  MoveL 10820 to (-38.97, 156.79, 153.89) mm, rotated rx -180 ry 0 rz 180 deg; joints [-53.214, -19.541, 102.145, 84.502, 53.57, -80.793]
  Call Extruder(791.10708)
  Set speed (40.0 mm/s)
  MoveL 10821 to (-38.97, 156.79, 153.89) mm, rotated rx -180 ry 0 rz 180 deg; joints [-53.214, -19.541, 102.145, 84.502, 53.57, -80.793]
  Call Extruder(0.00000)
  Set speed (130.0 mm/s)
  MoveL 10822 to (-31.64, 163.21, 153.89) mm, rotated rx 180 ry 0 rz 180 deg; joints [-52.884, -18.131, 101.16, 84.753, 53.204, -81.283]
  Call Extruder(2.00000)
  Set speed (40.0 mm/s)
  MoveL 10823 to (-31.64, 163.21, 153.89) mm, rotated rx 180 ry 0 rz 180 deg; joints [-52.884, -18.131, 101.16, 84.753, 53.204, -81.283]
  Set speed (30.0 mm/s)
  MoveL 10824 to (-31.64, 163.21, 153.89) mm, rotated rx 180 ry 0 rz 180 deg; joints [-52.884, -18.131, 101.16, 84.753, 53.204, -81.283]
  Call Extruder(2.18198)
  MoveL 10825 to (-31.93, 163.09, 153.89) mm, rotated rx 180 ry 0 rz 180 deg; joints [-52.91, -18.171, 101.189, 84.749, 53.231, -81.271]
  MoveL 10826 to (-31.93, 163.09, 153.89) mm, rotated rx 180 ry 0 rz 180 deg; joints [-52.91, -18.171, 101.189, 84.749, 53.231, -81.271]
  Call Extruder(2.36471)
  MoveL 10827 to (-32.22, 162.97, 153.89) mm, rotated rx -180 ry 0 rz -180 deg; joints [-52.936, -18.212, 101.218, 84.745, 53.257, -81.26]
  MoveL 10828 to (-32.22, 162.97, 153.89) mm, rotated rx -180 ry 0 rz -180 deg; joints [-52.936, -18.212, 101.218, 84.745, 53.257, -81.26]
  Call Extruder(2.53265)
  MoveL 10829 to (-32.49, 162.85, 153.89) mm, rotated rx 180 ry 0 rz 180 deg; joints [-52.96, -18.249, 101.244, 84.742, 53.282, -81.249]
  MoveL 10830 to (-32.49, 162.85, 153.89) mm, rotated rx 180 ry 0 rz 180 deg; joints [-52.96, -18.249, 101.244, 84.742, 53.282, -81.249]
  Call Extruder(2.68564)
  MoveL 10831 to (-32.73, 162.75, 153.89) mm, rotated rx -180 ry 0 rz 180 deg; joints [-52.981, -18.282, 101.268, 84.738, 53.304, -81.239]
  MoveL 10832 to (-32.73, 162.75, 153.89) mm, rotated rx -180 ry 0 rz 180 deg; joints [-52.981, -18.282, 101.268, 84.738, 53.304, -81.239]
  Call Extruder(2.83919)
  MoveL 10833 to (-32.97, 162.65, 153.89) mm, rotated rx 180 ry 0 rz 180 deg; joints [-53.002, -18.316, 101.292, 84.735, 53.326, -81.229]
  MoveL 10834 to (-32.97, 162.65, 153.89) mm, rotated rx 180 ry 0 rz 180 deg; joints [-53.002, -18.316, 101.292, 84.735, 53.326, -81.229]
  Call Extruder(3.04828)
  MoveL 10835 to (-33.28, 162.47, 153.89) mm, rotated rx -180 ry 0 rz 180 deg; joints [-53.025, -18.365, 101.326, 84.729, 53.349, -81.214]
  MoveL 10836 to (-33.28, 162.47, 153.89) mm, rotated rx -180 ry 0 rz 180 deg; joints [-53.025, -18.365, 101.326, 84.729, 53.349, -81.214]
  Call Extruder(3.25817)
  MoveL 10837 to (-33.59, 162.29, 153.89) mm, rotated rx 180 ry 0 rz 180 deg; joints [-53.048, -18.413, 101.36, 84.723, 53.373, -81.199]
  MoveL 10838 to (-33.59, 162.29, 153.89) mm, rotated rx 180 ry 0 rz 180 deg; joints [-53.048, -18.413, 101.36, 84.723, 53.373, -81.199]
  Call Extruder(3.46884)
  MoveL 10839 to (-33.9, 162.11, 153.89) mm, rotated rx 180 ry 0 rz 180 deg; joints [-53.07, -18.462, 101.394, 84.716, 53.397, -81.184]
  MoveL 10840 to (-33.9, 162.11, 153.89) mm, rotated rx 180 ry 0 rz 180 deg; joints [-53.07, -18.462, 101.394, 84.716, 53.397, -81.184]
  Call Extruder(3.68030)
  MoveL 10841 to (-34.2, 161.93, 153.89) mm, rotated rx -180 ry 0 rz 180 deg; joints [-53.093, -18.51, 101.428, 84.71, 53.421, -81.169]
  MoveL 10842 to (-34.2, 161.93, 153.89) mm, rotated rx -180 ry 0 rz 180 deg; joints [-53.093, -18.51, 101.428, 84.71, 53.421, -81.169]
  Call Extruder(3.88506)
  MoveL 10843 to (-34.49, 161.74, 153.89) mm, rotated rx 180 ry 0 rz -180 deg; joints [-53.111, -18.558, 101.462, 84.703, 53.439, -81.153]
  MoveL 10844 to (-34.49, 161.74, 153.89) mm, rotated rx 180 ry 0 rz -180 deg; joints [-53.111, -18.558, 101.462, 84.703, 53.439, -81.153]
  Call Extruder(4.20602)
  MoveL 10845 to (-34.92, 161.42, 153.89) mm, rotated rx 180 ry 0 rz 180 deg; joints [-53.137, -18.634, 101.516, 84.691, 53.467, -81.128]
  MoveL 10846 to (-34.92, 161.42, 153.89) mm, rotated rx 180 ry 0 rz 180 deg; joints [-53.137, -18.634, 101.516, 84.691, 53.467, -81.128]
  Call Extruder(4.52807)
  MoveL 10847 to (-35.35, 161.1, 153.89) mm, rotated rx 180 ry 0 rz -180 deg; joints [-53.163, -18.71, 101.569, 84.679, 53.495, -81.103]
  Call Extruder(5.35599)
  MoveL 10848 to (-36.39, 160.19, 153.89) mm, rotated rx 180 ry 0 rz 180 deg; joints [-53.209, -18.91, 101.708, 84.644, 53.547, -81.033]
  Call Extruder(6.18392)
  MoveL 10849 to (-37.3, 159.15, 153.89) mm, rotated rx -180 ry 0 rz 180 deg; joints [-53.227, -19.113, 101.85, 84.602, 53.57, -80.959]
  Call Extruder(6.34862)
  MoveL 10850 to (-37.46, 158.93, 153.89) mm, rotated rx -180 ry 0 rz 180 deg; joints [-53.227, -19.154, 101.878, 84.593, 53.571, -80.943]
  MoveL 10851 to (-37.46, 158.93, 153.89) mm, rotated rx -180 ry 0 rz 180 deg; joints [-53.227, -19.154, 101.878, 84.593, 53.571, -80.943]
  Call Extruder(6.67688)
  MoveL 10852 to (-37.79, 158.49, 153.89) mm, rotated rx -180 ry 0 rz 180 deg; joints [-53.226, -19.235, 101.934, 84.574, 53.572, -80.912]
  MoveL 10853 to (-37.79, 158.49, 153.89) mm, rotated rx -180 ry 0 rz 180 deg; joints [-53.226, -19.235, 101.934, 84.574, 53.572, -80.912]
  Call Extruder(7.00398)
  MoveL 10854 to (-38.11, 158.04, 153.89) mm, rotated rx 180 ry 0 rz 180 deg; joints [-53.224, -19.316, 101.99, 84.556, 53.573, -80.881]
  MoveL 10855 to (-38.11, 158.04, 153.89) mm, rotated rx 180 ry 0 rz 180 deg; joints [-53.224, -19.316, 101.99, 84.556, 53.573, -80.881]
  Call Extruder(7.13851)
  MoveL 10856 to (-38.23, 157.85, 153.89) mm, rotated rx -180 ry 0 rz 180 deg; joints [-53.22, -19.35, 102.013, 84.547, 53.57, -80.868]
  MoveL 10857 to (-38.23, 157.85, 153.89) mm, rotated rx -180 ry 0 rz 180 deg; joints [-53.22, -19.35, 102.013, 84.547, 53.57, -80.868]
  Call Extruder(7.35382)
  MoveL 10858 to (-38.41, 157.53, 153.89) mm, rotated rx 180 ry 0 rz 180 deg; joints [-53.213, -19.403, 102.05, 84.534, 53.564, -80.847]
  MoveL 10859 to (-38.41, 157.53, 153.89) mm, rotated rx 180 ry 0 rz 180 deg; joints [-53.213, -19.403, 102.05, 84.534, 53.564, -80.847]
  Call Extruder(7.56829)
  MoveL 10860 to (-38.59, 157.22, 153.89) mm, rotated rx 180 ry 0 rz 180 deg; joints [-53.205, -19.456, 102.087, 84.52, 53.559, -80.825]
  MoveL 10861 to (-38.59, 157.22, 153.89) mm, rotated rx 180 ry 0 rz 180 deg; joints [-53.205, -19.456, 102.087, 84.52, 53.559, -80.825]
  Call Extruder(7.78192)
  MoveL 10862 to (-38.77, 156.9, 153.89) mm, rotated rx 180 ry 0 rz 180 deg; joints [-53.198, -19.51, 102.123, 84.506, 53.553, -80.804]
  MoveL 10863 to (-38.77, 156.9, 153.89) mm, rotated rx 180 ry 0 rz 180 deg; joints [-53.198, -19.51, 102.123, 84.506, 53.553, -80.804]
  Call Extruder(7.96114)
  MoveL 10864 to (-38.91, 156.63, 153.89) mm, rotated rx 180 ry 0 rz 180 deg; joints [-53.189, -19.554, 102.154, 84.494, 53.546, -80.786]
  MoveL 10865 to (-38.91, 156.63, 153.89) mm, rotated rx 180 ry 0 rz 180 deg; joints [-53.189, -19.554, 102.154, 84.494, 53.546, -80.786]
  Call Extruder(8.10685)
  MoveL 10866 to (-39.01, 156.4, 153.89) mm, rotated rx -180 ry 0 rz 180 deg; joints [-53.18, -19.59, 102.179, 84.484, 53.537, -80.771]
  MoveL 10867 to (-39.01, 156.4, 153.89) mm, rotated rx -180 ry 0 rz 180 deg; joints [-53.18, -19.59, 102.179, 84.484, 53.537, -80.771]
  Call Extruder(8.25205)
  MoveL 10868 to (-39.1, 156.17, 153.89) mm, rotated rx -180 ry 0 rz 180 deg; joints [-53.17, -19.626, 102.203, 84.474, 53.528, -80.755]
  MoveL 10869 to (-39.1, 156.17, 153.89) mm, rotated rx -180 ry 0 rz 180 deg; joints [-53.17, -19.626, 102.203, 84.474, 53.528, -80.755]
  Call Extruder(8.43477)
  MoveL 10870 to (-39.23, 155.88, 153.89) mm, rotated rx 180 ry 0 rz 180 deg; joints [-53.156, -19.671, 102.234, 84.461, 53.517, -80.736]
  MoveL 10871 to (-39.23, 155.88, 153.89) mm, rotated rx 180 ry 0 rz 180 deg; joints [-53.156, -19.671, 102.234, 84.461, 53.517, -80.736]
  Call Extruder(8.61673)
  MoveL 10872 to (-39.35, 155.58, 153.89) mm, rotated rx 180 ry 0 rz 180 deg; joints [-53.143, -19.716, 102.265, 84.448, 53.505, -80.717]
  MoveL 10873 to (-39.35, 155.58, 153.89) mm, rotated rx 180 ry 0 rz 180 deg; joints [-53.143, -19.716, 102.265, 84.448, 53.505, -80.717]
  Call Extruder(8.76407)
  MoveL 10874 to (-39.44, 155.34, 153.89) mm, rotated rx 180 ry 0 rz -180 deg; joints [-53.131, -19.753, 102.29, 84.437, 53.495, -80.701]
  MoveL 10875 to (-39.44, 155.34, 153.89) mm, rotated rx 180 ry 0 rz -180 deg; joints [-53.131, -19.753, 102.29, 84.437, 53.495, -80.701]
  Call Extruder(8.87730)
  MoveL 10876 to (-39.5, 155.15, 153.89) mm, rotated rx 180 ry 0 rz -180 deg; joints [-53.121, -19.78, 102.309, 84.428, 53.485, -80.689]
  MoveL 10877 to (-39.5, 155.15, 153.89) mm, rotated rx 180 ry 0 rz -180 deg; joints [-53.121, -19.78, 102.309, 84.428, 53.485, -80.689]
  Call Extruder(8.99009)
  MoveL 10878 to (-39.56, 154.97, 153.89) mm, rotated rx 180 ry 0 rz 180 deg; joints [-53.11, -19.808, 102.328, 84.419, 53.475, -80.677]
  MoveL 10879 to (-39.56, 154.97, 153.89) mm, rotated rx 180 ry 0 rz 180 deg; joints [-53.11, -19.808, 102.328, 84.419, 53.475, -80.677]
  Call Extruder(9.10244)
  MoveL 10880 to (-39.62, 154.78, 153.89) mm, rotated rx 180 ry 0 rz 180 deg; joints [-53.099, -19.836, 102.347, 84.411, 53.465, -80.665]
  MoveL 10881 to (-39.62, 154.78, 153.89) mm, rotated rx 180 ry 0 rz 180 deg; joints [-53.099, -19.836, 102.347, 84.411, 53.465, -80.665]
  Call Extruder(9.21434)
  MoveL 10882 to (-39.68, 154.59, 153.89) mm, rotated rx 180 ry 0 rz 180 deg; joints [-53.088, -19.863, 102.366, 84.402, 53.455, -80.653]
  MoveL 10883 to (-39.68, 154.59, 153.89) mm, rotated rx 180 ry 0 rz 180 deg; joints [-53.088, -19.863, 102.366, 84.402, 53.455, -80.653]
  Call Extruder(9.33574)
  MoveL 10884 to (-39.75, 154.38, 153.89) mm, rotated rx -180 ry 0 rz 180 deg; joints [-53.076, -19.893, 102.386, 84.393, 53.444, -80.639]
  MoveL 10885 to (-39.75, 154.38, 153.89) mm, rotated rx -180 ry 0 rz 180 deg; joints [-53.076, -19.893, 102.386, 84.393, 53.444, -80.639]
  Call Extruder(9.46653)
  MoveL 10886 to (-39.81, 154.16, 153.89) mm, rotated rx 180 ry 0 rz 180 deg; joints [-53.063, -19.926, 102.408, 84.382, 53.432, -80.625]
  MoveL 10887 to (-39.81, 154.16, 153.89) mm, rotated rx 180 ry 0 rz 180 deg; joints [-53.063, -19.926, 102.408, 84.382, 53.432, -80.625]
  Call Extruder(9.59676)
  MoveL 10888 to (-39.88, 153.94, 153.89) mm, rotated rx 180 ry 0 rz -180 deg; joints [-53.049, -19.958, 102.43, 84.372, 53.42, -80.611]
  MoveL 10889 to (-39.88, 153.94, 153.89) mm, rotated rx 180 ry 0 rz -180 deg; joints [-53.049, -19.958, 102.43, 84.372, 53.42, -80.611]
  Call Extruder(9.72643)
  MoveL 10890 to (-39.95, 153.71, 153.89) mm, rotated rx 180 ry 0 rz 180 deg; joints [-53.036, -19.99, 102.452, 84.362, 53.407, -80.596]
  MoveL 10891 to (-39.95, 153.71, 153.89) mm, rotated rx 180 ry 0 rz 180 deg; joints [-53.036, -19.99, 102.452, 84.362, 53.407, -80.596]
  Call Extruder(9.85553)
  MoveL 10892 to (-40.02, 153.49, 153.89) mm, rotated rx 180 ry 0 rz 180 deg; joints [-53.022, -20.023, 102.474, 84.351, 53.395, -80.582]
  MoveL 10893 to (-40.02, 153.49, 153.89) mm, rotated rx 180 ry 0 rz 180 deg; joints [-53.022, -20.023, 102.474, 84.351, 53.395, -80.582]
  Call Extruder(9.97061)
  MoveL 10894 to (-40.06, 153.28, 153.89) mm, rotated rx -180 ry 0 rz 180 deg; joints [-53.007, -20.051, 102.493, 84.341, 53.381, -80.569]
  MoveL 10895 to (-40.06, 153.28, 153.89) mm, rotated rx -180 ry 0 rz 180 deg; joints [-53.007, -20.051, 102.493, 84.341, 53.381, -80.569]
  Call Extruder(10.08525)
  MoveL 10896 to (-40.11, 153.08, 153.89) mm, rotated rx -180 ry 0 rz 180 deg; joints [-52.993, -20.079, 102.512, 84.332, 53.368, -80.556]
  MoveL 10897 to (-40.11, 153.08, 153.89) mm, rotated rx -180 ry 0 rz 180 deg; joints [-52.993, -20.079, 102.512, 84.332, 53.368, -80.556]
  Call Extruder(10.19943)
  MoveL 10898 to (-40.15, 152.88, 153.89) mm, rotated rx 180 ry 0 rz 180 deg; joints [-52.978, -20.107, 102.531, 84.322, 53.354, -80.543]
  MoveL 10899 to (-40.15, 152.88, 153.89) mm, rotated rx 180 ry 0 rz 180 deg; joints [-52.978, -20.107, 102.531, 84.322, 53.354, -80.543]
  Call Extruder(10.31316)
  MoveL 10900 to (-40.2, 152.67, 153.89) mm, rotated rx 180 ry 0 rz -180 deg; joints [-52.963, -20.135, 102.55, 84.312, 53.34, -80.53]
  MoveL 10901 to (-40.2, 152.67, 153.89) mm, rotated rx 180 ry 0 rz -180 deg; joints [-52.963, -20.135, 102.55, 84.312, 53.34, -80.53]
  Call Extruder(10.43859)
  MoveL 10902 to (-40.24, 152.45, 153.89) mm, rotated rx -180 ry 0 rz 180 deg; joints [-52.946, -20.166, 102.571, 84.302, 53.325, -80.515]
  MoveL 10903 to (-40.24, 152.45, 153.89) mm, rotated rx -180 ry 0 rz 180 deg; joints [-52.946, -20.166, 102.571, 84.302, 53.325, -80.515]
  Call Extruder(10.57556)
  MoveL 10904 to (-40.29, 152.2, 153.89) mm, rotated rx -180 ry 0 rz 180 deg; joints [-52.928, -20.199, 102.594, 84.29, 53.308, -80.5]
  MoveL 10905 to (-40.29, 152.2, 153.89) mm, rotated rx -180 ry 0 rz 180 deg; joints [-52.928, -20.199, 102.594, 84.29, 53.308, -80.5]
  Call Extruder(10.71193)
  MoveL 10906 to (-40.34, 151.95, 153.89) mm, rotated rx 180 ry 0 rz 180 deg; joints [-52.909, -20.233, 102.617, 84.278, 53.29, -80.484]
  MoveL 10907 to (-40.34, 151.95, 153.89) mm, rotated rx 180 ry 0 rz 180 deg; joints [-52.909, -20.233, 102.617, 84.278, 53.29, -80.484]
  Call Extruder(10.84768)
  MoveL 10908 to (-40.39, 151.7, 153.89) mm, rotated rx -180 ry 0 rz 180 deg; joints [-52.89, -20.267, 102.639, 84.266, 53.273, -80.468]
  MoveL 10909 to (-40.39, 151.7, 153.89) mm, rotated rx -180 ry 0 rz 180 deg; joints [-52.89, -20.267, 102.639, 84.266, 53.273, -80.468]
  Call Extruder(10.98283)
  MoveL 10910 to (-40.44, 151.45, 153.89) mm, rotated rx -180 ry 0 rz 180 deg; joints [-52.871, -20.3, 102.662, 84.254, 53.255, -80.452]
  MoveL 10911 to (-40.44, 151.45, 153.89) mm, rotated rx -180 ry 0 rz 180 deg; joints [-52.871, -20.3, 102.662, 84.254, 53.255, -80.452]
  Call Extruder(11.11736)
  MoveL 10912 to (-40.49, 151.2, 153.89) mm, rotated rx 180 ry 0 rz 180 deg; joints [-52.853, -20.334, 102.685, 84.242, 53.238, -80.436]
  MoveL 10913 to (-40.49, 151.2, 153.89) mm, rotated rx 180 ry 0 rz 180 deg; joints [-52.853, -20.334, 102.685, 84.242, 53.238, -80.436]
  Call Extruder(11.25129)
  MoveL 10914 to (-40.54, 150.95, 153.89) mm, rotated rx 180 ry 0 rz 180 deg; joints [-52.834, -20.368, 102.707, 84.23, 53.22, -80.42]
  MoveL 10915 to (-40.54, 150.95, 153.89) mm, rotated rx 180 ry 0 rz 180 deg; joints [-52.834, -20.368, 102.707, 84.23, 53.22, -80.42]
  Call Extruder(11.39914)
  MoveL 10916 to (-40.59, 150.67, 153.89) mm, rotated rx 180 ry 0 rz 180 deg; joints [-52.812, -20.404, 102.732, 84.216, 53.2, -80.402]
  MoveL 10917 to (-40.59, 150.67, 153.89) mm, rotated rx 180 ry 0 rz 180 deg; joints [-52.812, -20.404, 102.732, 84.216, 53.2, -80.402]
  Call Extruder(11.56087)
  MoveL 10918 to (-40.64, 150.37, 153.89) mm, rotated rx 180 ry 0 rz 180 deg; joints [-52.787, -20.445, 102.759, 84.201, 53.177, -80.383]
  MoveL 10919 to (-40.64, 150.37, 153.89) mm, rotated rx 180 ry 0 rz 180 deg; joints [-52.787, -20.445, 102.759, 84.201, 53.177, -80.383]
  Call Extruder(11.72186)
  MoveL 10920 to (-40.69, 150.06, 153.89) mm, rotated rx 180 ry 0 rz 180 deg; joints [-52.762, -20.485, 102.786, 84.186, 53.154, -80.363]
  MoveL 10921 to (-40.69, 150.06, 153.89) mm, rotated rx 180 ry 0 rz 180 deg; joints [-52.762, -20.485, 102.786, 84.186, 53.154, -80.363]
  Call Extruder(11.88213)
  MoveL 10922 to (-40.73, 149.76, 153.89) mm, rotated rx -180 ry 0 rz 180 deg; joints [-52.737, -20.525, 102.813, 84.171, 53.13, -80.344]
  MoveL 10923 to (-40.73, 149.76, 153.89) mm, rotated rx -180 ry 0 rz 180 deg; joints [-52.737, -20.525, 102.813, 84.171, 53.13, -80.344]
  Call Extruder(12.04168)
  MoveL 10924 to (-40.78, 149.45, 153.89) mm, rotated rx -180 ry 0 rz 180 deg; joints [-52.712, -20.565, 102.84, 84.156, 53.107, -80.324]
  MoveL 10925 to (-40.78, 149.45, 153.89) mm, rotated rx -180 ry 0 rz 180 deg; joints [-52.712, -20.565, 102.84, 84.156, 53.107, -80.324]
  Call Extruder(12.20049)
  MoveL 10926 to (-40.83, 149.14, 153.89) mm, rotated rx 180 ry 0 rz 180 deg; joints [-52.687, -20.605, 102.867, 84.141, 53.084, -80.305]
  MoveL 10927 to (-40.83, 149.14, 153.89) mm, rotated rx 180 ry 0 rz 180 deg; joints [-52.687, -20.605, 102.867, 84.141, 53.084, -80.305]
  Call Extruder(12.37915)
  MoveL 10928 to (-40.88, 148.8, 153.89) mm, rotated rx 180 ry 0 rz 180 deg; joints [-52.658, -20.65, 102.897, 84.123, 53.056, -80.282]
  MoveL 10929 to (-40.88, 148.8, 153.89) mm, rotated rx 180 ry 0 rz 180 deg; joints [-52.658, -20.65, 102.897, 84.123, 53.056, -80.282]
  Call Extruder(12.57759)
  MoveL 10930 to (-40.92, 148.41, 153.89) mm, rotated rx 180 ry 0 rz 180 deg; joints [-52.624, -20.7, 102.93, 84.104, 53.024, -80.258]
  MoveL 10931 to (-40.92, 148.41, 153.89) mm, rotated rx 180 ry 0 rz 180 deg; joints [-52.624, -20.7, 102.93, 84.104, 53.024, -80.258]
  Call Extruder(12.77517)
  MoveL 10932 to (-40.97, 148.02, 153.89) mm, rotated rx 180 ry 0 rz -180 deg; joints [-52.59, -20.749, 102.963, 84.085, 52.993, -80.233]
  MoveL 10933 to (-40.97, 148.02, 153.89) mm, rotated rx 180 ry 0 rz -180 deg; joints [-52.59, -20.749, 102.963, 84.085, 52.993, -80.233]
  Call Extruder(12.97187)
  MoveL 10934 to (-41.02, 147.64, 153.89) mm, rotated rx 180 ry 0 rz 180 deg; joints [-52.556, -20.798, 102.996, 84.065, 52.961, -80.208]
  MoveL 10935 to (-41.02, 147.64, 153.89) mm, rotated rx 180 ry 0 rz 180 deg; joints [-52.556, -20.798, 102.996, 84.065, 52.961, -80.208]
  Call Extruder(13.16771)
  MoveL 10936 to (-41.06, 147.25, 153.89) mm, rotated rx -180 ry 0 rz 180 deg; joints [-52.521, -20.848, 103.029, 84.045, 52.929, -80.183]
  MoveL 10937 to (-41.06, 147.25, 153.89) mm, rotated rx -180 ry 0 rz 180 deg; joints [-52.521, -20.848, 103.029, 84.045, 52.929, -80.183]
  Call Extruder(13.46311)
  MoveL 10938 to (-41.11, 146.66, 153.89) mm, rotated rx 180 ry 0 rz -180 deg; joints [-52.466, -20.921, 103.078, 84.015, 52.877, -80.146]
  MoveL 10939 to (-41.11, 146.66, 153.89) mm, rotated rx 180 ry 0 rz -180 deg; joints [-52.466, -20.921, 103.078, 84.015, 52.877, -80.146]
  Call Extruder(13.75718)
  MoveL 10940 to (-41.15, 146.07, 153.89) mm, rotated rx 180 ry 0 rz 180 deg; joints [-52.411, -20.994, 103.126, 83.985, 52.825, -80.108]
  MoveL 10941 to (-41.15, 146.07, 153.89) mm, rotated rx 180 ry 0 rz 180 deg; joints [-52.411, -20.994, 103.126, 83.985, 52.825, -80.108]
  Call Extruder(14.04991)
  MoveL 10942 to (-41.2, 145.48, 153.89) mm, rotated rx 180 ry 0 rz -180 deg; joints [-52.355, -21.067, 103.175, 83.954, 52.773, -80.07]
  MoveL 10943 to (-41.2, 145.48, 153.89) mm, rotated rx 180 ry 0 rz -180 deg; joints [-52.355, -21.067, 103.175, 83.954, 52.773, -80.07]
  Call Extruder(14.62336)
  MoveL 10944 to (-41.25, 144.32, 153.89) mm, rotated rx -180 ry 0 rz 180 deg; joints [-52.239, -21.206, 103.267, 83.893, 52.663, -79.996]
  MoveL 10945 to (-41.25, 144.32, 153.89) mm, rotated rx -180 ry 0 rz 180 deg; joints [-52.239, -21.206, 103.267, 83.893, 52.663, -79.996]
  Call Extruder(15.33742)
  MoveL 10946 to (-41.29, 142.86, 153.89) mm, rotated rx 180 ry 0 rz 180 deg; joints [-52.09, -21.379, 103.38, 83.816, 52.523, -79.902]
  Call Extruder(57.40821)
  MoveL 10947 to (-41.29, 57.14, 153.89) mm, rotated rx 180 ry 0 rz 180 deg; joints [-40.759, -30.462, 108.688, 76.682, 42.138, -72.295]
  Call Extruder(57.85446)
  MoveL 10948 to (-41.27, 56.23, 153.89) mm, rotated rx 180 ry 0 rz 180 deg; joints [-40.608, -30.545, 108.731, 76.569, 42.004, -72.185]
  MoveL 10949 to (-41.27, 56.23, 153.89) mm, rotated rx 180 ry 0 rz 180 deg; joints [-40.608, -30.545, 108.731, 76.569, 42.004, -72.185]
  Call Extruder(58.44013)
  MoveL 10950 to (-41.22, 55.04, 153.89) mm, rotated rx -180 ry 0 rz 180 deg; joints [-40.408, -30.65, 108.784, 76.421, 41.826, -72.041]
  MoveL 10951 to (-41.22, 55.04, 153.89) mm, rotated rx -180 ry 0 rz 180 deg; joints [-40.408, -30.65, 108.784, 76.421, 41.826, -72.041]
  Call Extruder(58.87777)
  MoveL 10952 to (-41.17, 54.16, 153.89) mm, rotated rx 180 ry 0 rz 180 deg; joints [-40.257, -30.727, 108.823, 76.31, 41.691, -71.933]
  MoveL 10953 to (-41.17, 54.16, 153.89) mm, rotated rx 180 ry 0 rz 180 deg; joints [-40.257, -30.727, 108.823, 76.31, 41.691, -71.933]
  Call Extruder(59.16609)
  MoveL 10954 to (-41.13, 53.58, 153.89) mm, rotated rx -180 ry 0 rz 180 deg; joints [-40.156, -30.776, 108.848, 76.236, 41.6, -71.862]
  MoveL 10955 to (-41.13, 53.58, 153.89) mm, rotated rx -180 ry 0 rz 180 deg; joints [-40.156, -30.776, 108.848, 76.236, 41.6, -71.862]
  Call Extruder(59.45571)
  MoveL 10956 to (-41.08, 53, 153.89) mm, rotated rx 180 ry 0 rz 180 deg; joints [-40.054, -30.824, 108.872, 76.162, 41.51, -71.792]
  MoveL 10957 to (-41.08, 53, 153.89) mm, rotated rx 180 ry 0 rz 180 deg; joints [-40.054, -30.824, 108.872, 76.162, 41.51, -71.792]
  Call Extruder(59.69701)
  MoveL 10958 to (-41.04, 52.53, 153.89) mm, rotated rx -180 ry 0 rz -180 deg; joints [-39.969, -30.864, 108.892, 76.1, 41.433, -71.733]
  MoveL 10959 to (-41.04, 52.53, 153.89) mm, rotated rx -180 ry 0 rz -180 deg; joints [-39.969, -30.864, 108.892, 76.1, 41.433, -71.733]
  Call Extruder(59.88962)
  MoveL 10960 to (-40.99, 52.15, 153.89) mm, rotated rx 180 ry 0 rz -180 deg; joints [-39.9, -30.894, 108.907, 76.051, 41.371, -71.686]
  MoveL 10961 to (-40.99, 52.15, 153.89) mm, rotated rx 180 ry 0 rz -180 deg; joints [-39.9, -30.894, 108.907, 76.051, 41.371, -71.686]
  Call Extruder(60.08307)
  MoveL 10962 to (-40.95, 51.77, 153.89) mm, rotated rx 180 ry 0 rz 180 deg; joints [-39.83, -30.924, 108.922, 76.002, 41.309, -71.64]
  MoveL 10963 to (-40.95, 51.77, 153.89) mm, rotated rx 180 ry 0 rz 180 deg; joints [-39.83, -30.924, 108.922, 76.002, 41.309, -71.64]
  Call Extruder(60.27736)
  MoveL 10964 to (-40.9, 51.39, 153.89) mm, rotated rx 180 ry 0 rz 180 deg; joints [-39.761, -30.953, 108.937, 75.952, 41.247, -71.593]
  MoveL 10965 to (-40.9, 51.39, 153.89) mm, rotated rx 180 ry 0 rz 180 deg; joints [-39.761, -30.953, 108.937, 75.952, 41.247, -71.593]
  Call Extruder(60.47247)
  MoveL 10966 to (-40.86, 51.01, 153.89) mm, rotated rx -180 ry 0 rz 180 deg; joints [-39.692, -30.983, 108.952, 75.902, 41.185, -71.546]
  MoveL 10967 to (-40.86, 51.01, 153.89) mm, rotated rx -180 ry 0 rz 180 deg; joints [-39.692, -30.983, 108.952, 75.902, 41.185, -71.546]
  Call Extruder(60.63128)
  MoveL 10968 to (-40.81, 50.7, 153.89) mm, rotated rx -180 ry 0 rz 180 deg; joints [-39.634, -31.006, 108.964, 75.862, 41.133, -71.508]
  MoveL 10969 to (-40.81, 50.7, 153.89) mm, rotated rx -180 ry 0 rz 180 deg; joints [-39.634, -31.006, 108.964, 75.862, 41.133, -71.508]
  Call Extruder(60.79083)
  MoveL 10970 to (-40.76, 50.4, 153.89) mm, rotated rx 180 ry 0 rz 180 deg; joints [-39.576, -31.029, 108.975, 75.821, 41.081, -71.471]
  MoveL 10971 to (-40.76, 50.4, 153.89) mm, rotated rx 180 ry 0 rz 180 deg; joints [-39.576, -31.029, 108.975, 75.821, 41.081, -71.471]
  Call Extruder(60.95110)
  MoveL 10972 to (-40.71, 50.09, 153.89) mm, rotated rx 180 ry 0 rz 180 deg; joints [-39.518, -31.051, 108.986, 75.781, 41.029, -71.433]
  MoveL 10973 to (-40.71, 50.09, 153.89) mm, rotated rx 180 ry 0 rz 180 deg; joints [-39.518, -31.051, 108.986, 75.781, 41.029, -71.433]
  Call Extruder(61.11209)
  MoveL 10974 to (-40.66, 49.79, 153.89) mm, rotated rx 180 ry 0 rz -180 deg; joints [-39.46, -31.074, 108.998, 75.74, 40.976, -71.395]
  MoveL 10975 to (-40.66, 49.79, 153.89) mm, rotated rx 180 ry 0 rz -180 deg; joints [-39.46, -31.074, 108.998, 75.74, 40.976, -71.395]
  Call Extruder(61.27382)
  MoveL 10976 to (-40.61, 49.48, 153.89) mm, rotated rx -180 ry 0 rz 180 deg; joints [-39.402, -31.096, 109.009, 75.699, 40.924, -71.357]
  MoveL 10977 to (-40.61, 49.48, 153.89) mm, rotated rx -180 ry 0 rz 180 deg; joints [-39.402, -31.096, 109.009, 75.699, 40.924, -71.357]
  Call Extruder(61.43627)
  MoveL 10978 to (-40.57, 49.17, 153.89) mm, rotated rx 180 ry 0 rz 180 deg; joints [-39.344, -31.119, 109.02, 75.659, 40.872, -71.319]
  MoveL 10979 to (-40.57, 49.17, 153.89) mm, rotated rx 180 ry 0 rz 180 deg; joints [-39.344, -31.119, 109.02, 75.659, 40.872, -71.319]
  Call Extruder(61.57020)
  MoveL 10980 to (-40.52, 48.93, 153.89) mm, rotated rx 180 ry 0 rz 180 deg; joints [-39.296, -31.136, 109.029, 75.625, 40.828, -71.288]
  MoveL 10981 to (-40.52, 48.93, 153.89) mm, rotated rx 180 ry 0 rz 180 deg; joints [-39.296, -31.136, 109.029, 75.625, 40.828, -71.288]
  Call Extruder(61.70473)
  MoveL 10982 to (-40.47, 48.68, 153.89) mm, rotated rx 180 ry 0 rz 180 deg; joints [-39.247, -31.153, 109.037, 75.591, 40.784, -71.257]
  MoveL 10983 to (-40.47, 48.68, 153.89) mm, rotated rx 180 ry 0 rz 180 deg; joints [-39.247, -31.153, 109.037, 75.591, 40.784, -71.257]
  Call Extruder(61.83988)
  MoveL 10984 to (-40.42, 48.43, 153.89) mm, rotated rx -180 ry 0 rz 180 deg; joints [-39.198, -31.17, 109.046, 75.558, 40.74, -71.227]
  MoveL 10985 to (-40.42, 48.43, 153.89) mm, rotated rx -180 ry 0 rz 180 deg; joints [-39.198, -31.17, 109.046, 75.558, 40.74, -71.227]
  Call Extruder(61.97563)
  MoveL 10986 to (-40.37, 48.18, 153.89) mm, rotated rx -180 ry 0 rz 180 deg; joints [-39.149, -31.187, 109.054, 75.524, 40.696, -71.196]
  MoveL 10987 to (-40.37, 48.18, 153.89) mm, rotated rx -180 ry 0 rz 180 deg; joints [-39.149, -31.187, 109.054, 75.524, 40.696, -71.196]
  Call Extruder(62.11200)
  MoveL 10988 to (-40.32, 47.93, 153.89) mm, rotated rx -180 ry 0 rz 180 deg; joints [-39.1, -31.204, 109.063, 75.49, 40.652, -71.165]
  MoveL 10989 to (-40.32, 47.93, 153.89) mm, rotated rx -180 ry 0 rz 180 deg; joints [-39.1, -31.204, 109.063, 75.49, 40.652, -71.165]
  Call Extruder(62.24897)
  MoveL 10990 to (-40.27, 47.68, 153.89) mm, rotated rx 180 ry 0 rz 180 deg; joints [-39.051, -31.221, 109.071, 75.456, 40.607, -71.133]
  MoveL 10991 to (-40.27, 47.68, 153.89) mm, rotated rx 180 ry 0 rz 180 deg; joints [-39.051, -31.221, 109.071, 75.456, 40.607, -71.133]
  Call Extruder(62.38656)
  MoveL 10992 to (-40.22, 47.43, 153.89) mm, rotated rx 180 ry 0 rz -180 deg; joints [-39.002, -31.238, 109.08, 75.422, 40.563, -71.102]
  MoveL 10993 to (-40.22, 47.43, 153.89) mm, rotated rx 180 ry 0 rz -180 deg; joints [-39.002, -31.238, 109.08, 75.422, 40.563, -71.102]
  Call Extruder(62.50029)
  MoveL 10994 to (-40.17, 47.23, 153.89) mm, rotated rx -180 ry 0 rz 180 deg; joints [-38.962, -31.252, 109.087, 75.394, 40.526, -71.077]
  MoveL 10995 to (-40.17, 47.23, 153.89) mm, rotated rx -180 ry 0 rz 180 deg; joints [-38.962, -31.252, 109.087, 75.394, 40.526, -71.077]
  Call Extruder(62.61447)
  MoveL 10996 to (-40.13, 47.02, 153.89) mm, rotated rx -180 ry 0 rz 180 deg; joints [-38.921, -31.265, 109.093, 75.366, 40.489, -71.051]
  MoveL 10997 to (-40.13, 47.02, 153.89) mm, rotated rx -180 ry 0 rz 180 deg; joints [-38.921, -31.265, 109.093, 75.366, 40.489, -71.051]
  Call Extruder(62.72910)
  MoveL 10998 to (-40.08, 46.82, 153.89) mm, rotated rx 180 ry 0 rz -180 deg; joints [-38.88, -31.279, 109.1, 75.338, 40.452, -71.026]
  MoveL 10999 to (-40.08, 46.82, 153.89) mm, rotated rx 180 ry 0 rz -180 deg; joints [-38.88, -31.279, 109.1, 75.338, 40.452, -71.026]
  Call Extruder(62.84419)
  MoveL 11000 to (-40.04, 46.61, 153.89) mm, rotated rx 180 ry 0 rz 180 deg; joints [-38.839, -31.292, 109.107, 75.31, 40.416, -71]
  MoveL 11001 to (-40.04, 46.61, 153.89) mm, rotated rx 180 ry 0 rz 180 deg; joints [-38.839, -31.292, 109.107, 75.31, 40.416, -71]
  Call Extruder(62.96643)
  MoveL 11002 to (-39.98, 46.4, 153.89) mm, rotated rx -180 ry 0 rz -180 deg; joints [-38.795, -31.305, 109.113, 75.28, 40.376, -70.973]
  MoveL 11003 to (-39.98, 46.4, 153.89) mm, rotated rx -180 ry 0 rz -180 deg; joints [-38.795, -31.305, 109.113, 75.28, 40.376, -70.973]
  Call Extruder(63.09609)
  MoveL 11004 to (-39.92, 46.18, 153.89) mm, rotated rx 180 ry 0 rz 180 deg; joints [-38.748, -31.318, 109.119, 75.249, 40.332, -70.946]
  MoveL 11005 to (-39.92, 46.18, 153.89) mm, rotated rx 180 ry 0 rz 180 deg; joints [-38.748, -31.318, 109.119, 75.249, 40.332, -70.946]
  Call Extruder(63.22632)
  MoveL 11006 to (-39.85, 45.95, 153.89) mm, rotated rx 180 ry 0 rz 180 deg; joints [-38.7, -31.33, 109.125, 75.218, 40.289, -70.918]
  MoveL 11007 to (-39.85, 45.95, 153.89) mm, rotated rx 180 ry 0 rz 180 deg; joints [-38.7, -31.33, 109.125, 75.218, 40.289, -70.918]
  Call Extruder(63.35712)
  MoveL 11008 to (-39.78, 45.73, 153.89) mm, rotated rx 180 ry 0 rz 180 deg; joints [-38.653, -31.343, 109.132, 75.187, 40.246, -70.89]
  MoveL 11009 to (-39.78, 45.73, 153.89) mm, rotated rx 180 ry 0 rz 180 deg; joints [-38.653, -31.343, 109.132, 75.187, 40.246, -70.89]
  Call Extruder(63.48848)
  MoveL 11010 to (-39.71, 45.5, 153.89) mm, rotated rx -180 ry 0 rz 180 deg; joints [-38.605, -31.355, 109.138, 75.156, 40.203, -70.862]
  MoveL 11011 to (-39.71, 45.5, 153.89) mm, rotated rx -180 ry 0 rz 180 deg; joints [-38.605, -31.355, 109.138, 75.156, 40.203, -70.862]
  Call Extruder(63.60038)
  MoveL 11012 to (-39.65, 45.32, 153.89) mm, rotated rx 180 ry 0 rz 180 deg; joints [-38.565, -31.365, 109.143, 75.129, 40.166, -70.839]
  MoveL 11013 to (-39.65, 45.32, 153.89) mm, rotated rx 180 ry 0 rz 180 deg; joints [-38.565, -31.365, 109.143, 75.129, 40.166, -70.839]
  Call Extruder(63.71272)
  MoveL 11014 to (-39.59, 45.13, 153.89) mm, rotated rx 180 ry 0 rz 180 deg; joints [-38.524, -31.375, 109.148, 75.103, 40.129, -70.816]
  MoveL 11015 to (-39.59, 45.13, 153.89) mm, rotated rx 180 ry 0 rz 180 deg; joints [-38.524, -31.375, 109.148, 75.103, 40.129, -70.816]
  Call Extruder(63.82551)
  MoveL 11016 to (-39.53, 44.94, 153.89) mm, rotated rx 180 ry 0 rz 180 deg; joints [-38.483, -31.385, 109.153, 75.076, 40.092, -70.792]
  MoveL 11017 to (-39.53, 44.94, 153.89) mm, rotated rx 180 ry 0 rz 180 deg; joints [-38.483, -31.385, 109.153, 75.076, 40.092, -70.792]
  Call Extruder(63.93874)
  MoveL 11018 to (-39.47, 44.75, 153.89) mm, rotated rx -180 ry 0 rz 180 deg; joints [-38.443, -31.395, 109.158, 75.05, 40.054, -70.769]
  MoveL 11019 to (-39.47, 44.75, 153.89) mm, rotated rx -180 ry 0 rz 180 deg; joints [-38.443, -31.395, 109.158, 75.05, 40.054, -70.769]
  Call Extruder(64.05242)
  MoveL 11020 to (-39.41, 44.56, 153.89) mm, rotated rx -180 ry 0 rz 180 deg; joints [-38.402, -31.405, 109.163, 75.023, 40.017, -70.745]
  MoveL 11021 to (-39.41, 44.56, 153.89) mm, rotated rx -180 ry 0 rz 180 deg; joints [-38.402, -31.405, 109.163, 75.023, 40.017, -70.745]
  Call Extruder(64.23439)
  MoveL 11022 to (-39.29, 44.27, 153.89) mm, rotated rx 180 ry 0 rz 180 deg; joints [-38.335, -31.417, 109.169, 74.982, 39.956, -70.71]
  MoveL 11023 to (-39.29, 44.27, 153.89) mm, rotated rx 180 ry 0 rz 180 deg; joints [-38.335, -31.417, 109.169, 74.982, 39.956, -70.71]
  Call Extruder(64.41711)
  MoveL 11024 to (-39.16, 43.98, 153.89) mm, rotated rx 180 ry 0 rz 180 deg; joints [-38.269, -31.43, 109.175, 74.94, 39.895, -70.674]
  MoveL 11025 to (-39.16, 43.98, 153.89) mm, rotated rx 180 ry 0 rz 180 deg; joints [-38.269, -31.43, 109.175, 74.94, 39.895, -70.674]
  Call Extruder(64.58752)
  MoveL 11026 to (-39.05, 43.71, 153.89) mm, rotated rx 180 ry 0 rz -180 deg; joints [-38.207, -31.441, 109.18, 74.902, 39.838, -70.641]
  MoveL 11027 to (-39.05, 43.71, 153.89) mm, rotated rx 180 ry 0 rz -180 deg; joints [-38.207, -31.441, 109.18, 74.902, 39.838, -70.641]
  Call Extruder(64.74550)
  MoveL 11028 to (-38.94, 43.46, 153.89) mm, rotated rx 180 ry 0 rz 180 deg; joints [-38.149, -31.451, 109.185, 74.866, 39.785, -70.611]
  MoveL 11029 to (-38.94, 43.46, 153.89) mm, rotated rx 180 ry 0 rz 180 deg; joints [-38.149, -31.451, 109.185, 74.866, 39.785, -70.611]
  Call Extruder(64.90409)
  MoveL 11030 to (-38.84, 43.21, 153.89) mm, rotated rx 180 ry 0 rz 180 deg; joints [-38.092, -31.461, 109.19, 74.83, 39.732, -70.58]
  MoveL 11031 to (-38.84, 43.21, 153.89) mm, rotated rx 180 ry 0 rz 180 deg; joints [-38.092, -31.461, 109.19, 74.83, 39.732, -70.58]
  Call Extruder(65.11025)
  MoveL 11032 to (-38.66, 42.91, 153.89) mm, rotated rx -180 ry 0 rz 180 deg; joints [-38.016, -31.468, 109.194, 74.786, 39.661, -70.544]
  MoveL 11033 to (-38.66, 42.91, 153.89) mm, rotated rx -180 ry 0 rz 180 deg; joints [-38.016, -31.468, 109.194, 74.786, 39.661, -70.544]
  Call Extruder(65.31720)
  MoveL 11034 to (-38.49, 42.6, 153.89) mm, rotated rx -180 ry 0 rz -180 deg; joints [-37.939, -31.475, 109.197, 74.742, 39.59, -70.508]
  MoveL 11035 to (-38.49, 42.6, 153.89) mm, rotated rx -180 ry 0 rz -180 deg; joints [-37.939, -31.475, 109.197, 74.742, 39.59, -70.508]
  Call Extruder(65.52492)
  MoveL 11036 to (-38.31, 42.3, 153.89) mm, rotated rx 180 ry 0 rz -180 deg; joints [-37.863, -31.482, 109.201, 74.698, 39.519, -70.472]
  MoveL 11037 to (-38.31, 42.3, 153.89) mm, rotated rx 180 ry 0 rz -180 deg; joints [-37.863, -31.482, 109.201, 74.698, 39.519, -70.472]
  Call Extruder(65.73342)
  MoveL 11038 to (-38.13, 41.99, 153.89) mm, rotated rx 180 ry 0 rz 180 deg; joints [-37.787, -31.489, 109.204, 74.654, 39.448, -70.435]
  MoveL 11039 to (-38.13, 41.99, 153.89) mm, rotated rx 180 ry 0 rz 180 deg; joints [-37.787, -31.489, 109.204, 74.654, 39.448, -70.435]
  Call Extruder(65.91297)
  MoveL 11040 to (-37.96, 41.75, 153.89) mm, rotated rx 180 ry 0 rz 180 deg; joints [-37.72, -31.49, 109.205, 74.618, 39.386, -70.407]
  MoveL 11041 to (-37.96, 41.75, 153.89) mm, rotated rx 180 ry 0 rz 180 deg; joints [-37.72, -31.49, 109.205, 74.618, 39.386, -70.407]
  Call Extruder(66.24641)
  MoveL 11042 to (-37.63, 41.3, 153.89) mm, rotated rx 180 ry 0 rz 180 deg; joints [-37.598, -31.492, 109.206, 74.552, 39.271, -70.355]
  MoveL 11043 to (-37.63, 41.3, 153.89) mm, rotated rx 180 ry 0 rz 180 deg; joints [-37.598, -31.492, 109.206, 74.552, 39.271, -70.355]
  Call Extruder(66.58104)
  MoveL 11044 to (-37.3, 40.85, 153.89) mm, rotated rx -180 ry 0 rz 180 deg; joints [-37.475, -31.495, 109.207, 74.485, 39.156, -70.303]
  Call Extruder(67.40900)
  MoveL 11045 to (-36.39, 39.81, 153.89) mm, rotated rx -180 ry 0 rz 180 deg; joints [-37.173, -31.481, 109.2, 74.331, 38.869, -70.188]
  Call Extruder(68.06491)
  MoveL 11046 to (-35.57, 39.08, 153.89) mm, rotated rx 180 ry 0 rz 180 deg; joints [-36.937, -31.45, 109.185, 74.222, 38.643, -70.112]
  Call Extruder(68.40395)
  MoveL 11047 to (-35.13, 38.73, 153.89) mm, rotated rx 180 ry 0 rz 180 deg; joints [-36.818, -31.429, 109.174, 74.17, 38.528, -70.077]
  MoveL 11048 to (-35.13, 38.73, 153.89) mm, rotated rx 180 ry 0 rz 180 deg; joints [-36.818, -31.429, 109.174, 74.17, 38.528, -70.077]
  Call Extruder(68.73731)
  MoveL 11049 to (-34.68, 38.41, 153.89) mm, rotated rx 180 ry 0 rz 180 deg; joints [-36.701, -31.405, 109.163, 74.12, 38.415, -70.046]
  MoveL 11050 to (-34.68, 38.41, 153.89) mm, rotated rx 180 ry 0 rz 180 deg; joints [-36.701, -31.405, 109.163, 74.12, 38.415, -70.046]
  Call Extruder(69.06951)
  MoveL 11051 to (-34.22, 38.08, 153.89) mm, rotated rx 180 ry 0 rz 180 deg; joints [-36.584, -31.381, 109.151, 74.071, 38.302, -70.014]
  MoveL 11052 to (-34.22, 38.08, 153.89) mm, rotated rx 180 ry 0 rz 180 deg; joints [-36.584, -31.381, 109.151, 74.071, 38.302, -70.014]
  Call Extruder(69.24304)
  MoveL 11053 to (-33.97, 37.93, 153.89) mm, rotated rx 180 ry 0 rz 180 deg; joints [-36.525, -31.365, 109.143, 74.048, 38.244, -70.002]
  MoveL 11054 to (-33.97, 37.93, 153.89) mm, rotated rx 180 ry 0 rz 180 deg; joints [-36.525, -31.365, 109.143, 74.048, 38.244, -70.002]
  Call Extruder(69.46654)
  MoveL 11055 to (-33.64, 37.74, 153.89) mm, rotated rx 180 ry 0 rz 180 deg; joints [-36.449, -31.343, 109.132, 74.02, 38.17, -69.986]
  MoveL 11056 to (-33.64, 37.74, 153.89) mm, rotated rx 180 ry 0 rz 180 deg; joints [-36.449, -31.343, 109.132, 74.02, 38.17, -69.986]
  Call Extruder(69.68914)
  MoveL 11057 to (-33.32, 37.55, 153.89) mm, rotated rx 180 ry 0 rz 180 deg; joints [-36.374, -31.321, 109.121, 73.991, 38.096, -69.97]
  MoveL 11058 to (-33.32, 37.55, 153.89) mm, rotated rx 180 ry 0 rz 180 deg; joints [-36.374, -31.321, 109.121, 73.991, 38.096, -69.97]
  Call Extruder(69.91084)
  MoveL 11059 to (-32.99, 37.36, 153.89) mm, rotated rx 180 ry 0 rz 180 deg; joints [-36.298, -31.299, 109.11, 73.963, 38.022, -69.954]
  MoveL 11060 to (-32.99, 37.36, 153.89) mm, rotated rx 180 ry 0 rz 180 deg; joints [-36.298, -31.299, 109.11, 73.963, 38.022, -69.954]
  Call Extruder(70.07784)
  MoveL 11061 to (-32.73, 37.25, 153.89) mm, rotated rx 180 ry 0 rz 180 deg; joints [-36.244, -31.279, 109.1, 73.946, 37.968, -69.946]
  MoveL 11062 to (-32.73, 37.25, 153.89) mm, rotated rx 180 ry 0 rz 180 deg; joints [-36.244, -31.279, 109.1, 73.946, 37.968, -69.946]
  Call Extruder(70.24417)
  MoveL 11063 to (-32.46, 37.14, 153.89) mm, rotated rx -180 ry 0 rz 180 deg; joints [-36.19, -31.258, 109.09, 73.928, 37.915, -69.939]
  MoveL 11064 to (-32.46, 37.14, 153.89) mm, rotated rx -180 ry 0 rz 180 deg; joints [-36.19, -31.258, 109.09, 73.928, 37.915, -69.939]
  Call Extruder(70.41418)
  MoveL 11065 to (-32.19, 37.02, 153.89) mm, rotated rx 180 ry 0 rz 180 deg; joints [-36.135, -31.236, 109.079, 73.911, 37.86, -69.932]
  MoveL 11066 to (-32.19, 37.02, 153.89) mm, rotated rx 180 ry 0 rz 180 deg; joints [-36.135, -31.236, 109.079, 73.911, 37.86, -69.932]
  Call Extruder(70.58788)
  MoveL 11067 to (-31.91, 36.91, 153.89) mm, rotated rx -180 ry 0 rz -180 deg; joints [-36.079, -31.214, 109.068, 73.894, 37.804, -69.925]
  MoveL 11068 to (-31.91, 36.91, 153.89) mm, rotated rx -180 ry 0 rz -180 deg; joints [-36.079, -31.214, 109.068, 73.894, 37.804, -69.925]
  Call Extruder(70.76089)
  MoveL 11069 to (-31.64, 36.79, 153.89) mm, rotated rx 180 ry 0 rz 180 deg; joints [-36.023, -31.191, 109.056, 73.876, 37.749, -69.918]
  MoveL 11070 to (-31.64, 36.79, 153.89) mm, rotated rx 180 ry 0 rz 180 deg; joints [-36.023, -31.191, 109.056, 73.876, 37.749, -69.918]
  Call Extruder(70.87435)
  MoveL 11071 to (-31.45, 36.73, 153.89) mm, rotated rx 180 ry 0 rz 180 deg; joints [-35.989, -31.174, 109.048, 73.867, 37.713, -69.915]
  MoveL 11072 to (-31.45, 36.73, 153.89) mm, rotated rx 180 ry 0 rz 180 deg; joints [-35.989, -31.174, 109.048, 73.867, 37.713, -69.915]
  Call Extruder(70.98736)
  MoveL 11073 to (-31.26, 36.67, 153.89) mm, rotated rx 180 ry 0 rz 180 deg; joints [-35.954, -31.158, 109.04, 73.858, 37.678, -69.913]
  MoveL 11074 to (-31.26, 36.67, 153.89) mm, rotated rx 180 ry 0 rz 180 deg; joints [-35.954, -31.158, 109.04, 73.858, 37.678, -69.913]
  Call Extruder(71.09993)
  MoveL 11075 to (-31.07, 36.61, 153.89) mm, rotated rx 180 ry 0 rz 180 deg; joints [-35.919, -31.141, 109.031, 73.849, 37.643, -69.911]
  MoveL 11076 to (-31.07, 36.61, 153.89) mm, rotated rx 180 ry 0 rz 180 deg; joints [-35.919, -31.141, 109.031, 73.849, 37.643, -69.911]
  Call Extruder(71.21206)
  MoveL 11077 to (-30.88, 36.55, 153.89) mm, rotated rx 180 ry 0 rz -180 deg; joints [-35.884, -31.124, 109.023, 73.84, 37.608, -69.908]
  MoveL 11078 to (-30.88, 36.55, 153.89) mm, rotated rx 180 ry 0 rz -180 deg; joints [-35.884, -31.124, 109.023, 73.84, 37.608, -69.908]
  Call Extruder(71.32374)
  MoveL 11079 to (-30.7, 36.49, 153.89) mm, rotated rx 180 ry 0 rz 180 deg; joints [-35.849, -31.107, 109.014, 73.831, 37.573, -69.906]
  MoveL 11080 to (-30.7, 36.49, 153.89) mm, rotated rx 180 ry 0 rz 180 deg; joints [-35.849, -31.107, 109.014, 73.831, 37.573, -69.906]
  Call Extruder(71.45479)
  MoveL 11081 to (-30.47, 36.42, 153.89) mm, rotated rx 180 ry 0 rz 180 deg; joints [-35.809, -31.087, 109.004, 73.821, 37.532, -69.904]
  MoveL 11082 to (-30.47, 36.42, 153.89) mm, rotated rx 180 ry 0 rz 180 deg; joints [-35.809, -31.087, 109.004, 73.821, 37.532, -69.904]
  Call Extruder(71.58528)
  MoveL 11083 to (-30.25, 36.35, 153.89) mm, rotated rx 180 ry 0 rz 180 deg; joints [-35.769, -31.067, 108.994, 73.811, 37.492, -69.902]
  MoveL 11084 to (-30.25, 36.35, 153.89) mm, rotated rx 180 ry 0 rz 180 deg; joints [-35.769, -31.067, 108.994, 73.811, 37.492, -69.902]
  Call Extruder(71.71521)
  MoveL 11085 to (-30.02, 36.28, 153.89) mm, rotated rx 180 ry 0 rz -180 deg; joints [-35.728, -31.046, 108.984, 73.801, 37.451, -69.9]
  MoveL 11086 to (-30.02, 36.28, 153.89) mm, rotated rx 180 ry 0 rz -180 deg; joints [-35.728, -31.046, 108.984, 73.801, 37.451, -69.9]
  Call Extruder(71.84457)
  MoveL 11087 to (-29.8, 36.22, 153.89) mm, rotated rx -180 ry 0 rz 180 deg; joints [-35.688, -31.026, 108.974, 73.791, 37.41, -69.898]
  MoveL 11088 to (-29.8, 36.22, 153.89) mm, rotated rx -180 ry 0 rz 180 deg; joints [-35.688, -31.026, 108.974, 73.791, 37.41, -69.898]
  Call Extruder(71.96654)
  MoveL 11089 to (-29.59, 36.16, 153.89) mm, rotated rx 180 ry 0 rz -180 deg; joints [-35.651, -31.005, 108.963, 73.782, 37.373, -69.897]
  MoveL 11090 to (-29.59, 36.16, 153.89) mm, rotated rx 180 ry 0 rz -180 deg; joints [-35.651, -31.005, 108.963, 73.782, 37.373, -69.897]
  Call Extruder(72.08140)
  MoveL 11091 to (-29.38, 36.12, 153.89) mm, rotated rx 180 ry 0 rz 180 deg; joints [-35.617, -30.985, 108.953, 73.776, 37.339, -69.898]
  MoveL 11092 to (-29.38, 36.12, 153.89) mm, rotated rx 180 ry 0 rz 180 deg; joints [-35.617, -30.985, 108.953, 73.776, 37.339, -69.898]
  Call Extruder(72.19582)
  MoveL 11093 to (-29.18, 36.07, 153.89) mm, rotated rx 180 ry 0 rz 180 deg; joints [-35.584, -30.965, 108.943, 73.769, 37.304, -69.899]
  MoveL 11094 to (-29.18, 36.07, 153.89) mm, rotated rx 180 ry 0 rz 180 deg; joints [-35.584, -30.965, 108.943, 73.769, 37.304, -69.899]
  Call Extruder(72.30978)
  MoveL 11095 to (-28.97, 36.03, 153.89) mm, rotated rx 180 ry 0 rz 180 deg; joints [-35.55, -30.945, 108.933, 73.763, 37.27, -69.899]
  MoveL 11096 to (-28.97, 36.03, 153.89) mm, rotated rx 180 ry 0 rz 180 deg; joints [-35.55, -30.945, 108.933, 73.763, 37.27, -69.899]
  Call Extruder(72.42328)
  MoveL 11097 to (-28.77, 35.98, 153.89) mm, rotated rx 180 ry 0 rz 180 deg; joints [-35.517, -30.925, 108.923, 73.757, 37.236, -69.9]
  MoveL 11098 to (-28.77, 35.98, 153.89) mm, rotated rx 180 ry 0 rz 180 deg; joints [-35.517, -30.925, 108.923, 73.757, 37.236, -69.9]
  Call Extruder(72.56057)
  MoveL 11099 to (-28.52, 35.93, 153.89) mm, rotated rx 180 ry 0 rz 180 deg; joints [-35.477, -30.9, 108.91, 73.75, 37.194, -69.902]
  MoveL 11100 to (-28.52, 35.93, 153.89) mm, rotated rx 180 ry 0 rz 180 deg; joints [-35.477, -30.9, 108.91, 73.75, 37.194, -69.902]
  Call Extruder(72.69724)
  MoveL 11101 to (-28.27, 35.88, 153.89) mm, rotated rx -180 ry 0 rz 180 deg; joints [-35.437, -30.875, 108.898, 73.743, 37.154, -69.904]
  MoveL 11102 to (-28.27, 35.88, 153.89) mm, rotated rx -180 ry 0 rz 180 deg; joints [-35.437, -30.875, 108.898, 73.743, 37.154, -69.904]
  Call Extruder(72.83330)
  MoveL 11103 to (-28.02, 35.83, 153.89) mm, rotated rx 180 ry 0 rz 180 deg; joints [-35.397, -30.85, 108.885, 73.736, 37.113, -69.905]
  MoveL 11104 to (-28.02, 35.83, 153.89) mm, rotated rx 180 ry 0 rz 180 deg; joints [-35.397, -30.85, 108.885, 73.736, 37.113, -69.905]
  Call Extruder(72.96875)
  MoveL 11105 to (-27.77, 35.78, 153.89) mm, rotated rx 180 ry 0 rz 180 deg; joints [-35.357, -30.825, 108.873, 73.729, 37.072, -69.907]
  MoveL 11106 to (-27.77, 35.78, 153.89) mm, rotated rx 180 ry 0 rz 180 deg; joints [-35.357, -30.825, 108.873, 73.729, 37.072, -69.907]
  Call Extruder(73.10359)
  MoveL 11107 to (-27.52, 35.73, 153.89) mm, rotated rx 180 ry 0 rz 180 deg; joints [-35.317, -30.8, 108.86, 73.722, 37.031, -69.909]
  MoveL 11108 to (-27.52, 35.73, 153.89) mm, rotated rx 180 ry 0 rz 180 deg; joints [-35.317, -30.8, 108.86, 73.722, 37.031, -69.909]
  Call Extruder(73.23783)
  MoveL 11109 to (-27.28, 35.68, 153.89) mm, rotated rx 180 ry 0 rz 180 deg; joints [-35.277, -30.775, 108.847, 73.715, 36.99, -69.91]
  MoveL 11110 to (-27.28, 35.68, 153.89) mm, rotated rx 180 ry 0 rz 180 deg; joints [-35.277, -30.775, 108.847, 73.715, 36.99, -69.91]
  Call Extruder(73.37145)
  MoveL 11111 to (-27.02, 35.63, 153.89) mm, rotated rx -180 ry 0 rz 180 deg; joints [-35.238, -30.749, 108.834, 73.708, 36.949, -69.912]
  MoveL 11112 to (-27.02, 35.63, 153.89) mm, rotated rx -180 ry 0 rz 180 deg; joints [-35.238, -30.749, 108.834, 73.708, 36.949, -69.912]
  Call Extruder(73.53354)
  MoveL 11113 to (-26.72, 35.59, 153.89) mm, rotated rx 180 ry 0 rz 180 deg; joints [-35.191, -30.718, 108.818, 73.702, 36.901, -69.916]
  MoveL 11114 to (-26.72, 35.59, 153.89) mm, rotated rx 180 ry 0 rz 180 deg; joints [-35.191, -30.718, 108.818, 73.702, 36.901, -69.916]
  Call Extruder(73.69491)
  MoveL 11115 to (-26.41, 35.54, 153.89) mm, rotated rx -180 ry 0 rz 180 deg; joints [-35.145, -30.686, 108.802, 73.695, 36.853, -69.92]
  MoveL 11116 to (-26.41, 35.54, 153.89) mm, rotated rx -180 ry 0 rz 180 deg; joints [-35.145, -30.686, 108.802, 73.695, 36.853, -69.92]
  Call Extruder(73.85555)
  MoveL 11117 to (-26.11, 35.49, 153.89) mm, rotated rx -180 ry 0 rz 180 deg; joints [-35.098, -30.654, 108.786, 73.689, 36.805, -69.924]
  MoveL 11118 to (-26.11, 35.49, 153.89) mm, rotated rx -180 ry 0 rz 180 deg; joints [-35.098, -30.654, 108.786, 73.689, 36.805, -69.924]
  Call Extruder(74.01546)
  MoveL 11119 to (-25.8, 35.44, 153.89) mm, rotated rx 180 ry 0 rz 180 deg; joints [-35.052, -30.622, 108.77, 73.683, 36.757, -69.928]
  MoveL 11120 to (-25.8, 35.44, 153.89) mm, rotated rx 180 ry 0 rz 180 deg; joints [-35.052, -30.622, 108.77, 73.683, 36.757, -69.928]
  Call Extruder(74.17465)
  MoveL 11121 to (-25.5, 35.39, 153.89) mm, rotated rx 180 ry 0 rz 180 deg; joints [-35.006, -30.59, 108.754, 73.676, 36.71, -69.932]
  MoveL 11122 to (-25.5, 35.39, 153.89) mm, rotated rx 180 ry 0 rz 180 deg; joints [-35.006, -30.59, 108.754, 73.676, 36.71, -69.932]
  Call Extruder(74.33311)
  MoveL 11123 to (-25.19, 35.34, 153.89) mm, rotated rx 180 ry 0 rz 180 deg; joints [-34.96, -30.558, 108.737, 73.67, 36.662, -69.936]
  MoveL 11124 to (-25.19, 35.34, 153.89) mm, rotated rx 180 ry 0 rz 180 deg; joints [-34.96, -30.558, 108.737, 73.67, 36.662, -69.936]
  Call Extruder(74.53198)
  MoveL 11125 to (-24.8, 35.3, 153.89) mm, rotated rx 180 ry 0 rz 180 deg; joints [-34.904, -30.516, 108.716, 73.665, 36.604, -69.943]
  MoveL 11126 to (-24.8, 35.3, 153.89) mm, rotated rx 180 ry 0 rz 180 deg; joints [-34.904, -30.516, 108.716, 73.665, 36.604, -69.943]
  Call Extruder(74.72999)
  MoveL 11127 to (-24.42, 35.25, 153.89) mm, rotated rx -180 ry 0 rz 180 deg; joints [-34.849, -30.474, 108.694, 73.659, 36.546, -69.951]
  MoveL 11128 to (-24.42, 35.25, 153.89) mm, rotated rx -180 ry 0 rz 180 deg; joints [-34.849, -30.474, 108.694, 73.659, 36.546, -69.951]
  Call Extruder(74.92713)
  MoveL 11129 to (-24.03, 35.21, 153.89) mm, rotated rx -180 ry 0 rz -180 deg; joints [-34.794, -30.432, 108.673, 73.654, 36.488, -69.958]
  MoveL 11130 to (-24.03, 35.21, 153.89) mm, rotated rx -180 ry 0 rz -180 deg; joints [-34.794, -30.432, 108.673, 73.654, 36.488, -69.958]
  Call Extruder(75.12340)
  MoveL 11131 to (-23.64, 35.16, 153.89) mm, rotated rx 180 ry 0 rz 180 deg; joints [-34.739, -30.39, 108.651, 73.649, 36.431, -69.966]
  MoveL 11132 to (-23.64, 35.16, 153.89) mm, rotated rx 180 ry 0 rz 180 deg; joints [-34.739, -30.39, 108.651, 73.649, 36.431, -69.966]
  Call Extruder(75.36909)
  MoveL 11133 to (-23.15, 35.11, 153.89) mm, rotated rx 180 ry 0 rz 180 deg; joints [-34.671, -30.336, 108.624, 73.644, 36.36, -69.977]
  MoveL 11134 to (-23.15, 35.11, 153.89) mm, rotated rx 180 ry 0 rz 180 deg; joints [-34.671, -30.336, 108.624, 73.644, 36.36, -69.977]
  Call Extruder(75.66381)
  MoveL 11135 to (-22.56, 35.07, 153.89) mm, rotated rx 180 ry 0 rz -180 deg; joints [-34.592, -30.27, 108.59, 73.641, 36.276, -69.992]
  MoveL 11136 to (-22.56, 35.07, 153.89) mm, rotated rx 180 ry 0 rz -180 deg; joints [-34.592, -30.27, 108.59, 73.641, 36.276, -69.992]
  Call Extruder(75.95720)
  MoveL 11137 to (-21.97, 35.02, 153.89) mm, rotated rx 180 ry 0 rz 180 deg; joints [-34.512, -30.204, 108.556, 73.637, 36.193, -70.007]
  MoveL 11138 to (-21.97, 35.02, 153.89) mm, rotated rx 180 ry 0 rz 180 deg; joints [-34.512, -30.204, 108.556, 73.637, 36.193, -70.007]
  Call Extruder(76.39052)
  MoveL 11139 to (-21.1, 34.98, 153.89) mm, rotated rx 180 ry 0 rz -180 deg; joints [-34.399, -30.103, 108.504, 73.635, 36.073, -70.033]
  MoveL 11140 to (-21.1, 34.98, 153.89) mm, rotated rx 180 ry 0 rz -180 deg; joints [-34.399, -30.103, 108.504, 73.635, 36.073, -70.033]
  Call Extruder(76.96268)
  MoveL 11141 to (-19.94, 34.93, 153.89) mm, rotated rx 180 ry 0 rz -180 deg; joints [-34.253, -29.969, 108.435, 73.636, 35.917, -70.071]
  MoveL 11142 to (-19.94, 34.93, 153.89) mm, rotated rx 180 ry 0 rz -180 deg; joints [-34.253, -29.969, 108.435, 73.636, 35.917, -70.071]
  Call Extruder(77.39112)
  MoveL 11143 to (-19.06, 34.91, 153.89) mm, rotated rx 180 ry 0 rz 180 deg; joints [-34.146, -29.866, 108.381, 73.639, 35.803, -70.101]
  Call Extruder(194.20579)
  MoveL 11144 to (219.06, 34.92, 153.89) mm, rotated rx 180 ry 0 rz 180 deg; joints [-18.249, 2.515, 83.098, 76.94, 18.751, -76.235]
  Call Extruder(194.63413)
  MoveL 11145 to (219.93, 34.93, 153.89) mm, rotated rx 180 ry 0 rz 180 deg; joints [-18.219, 2.648, 82.959, 76.902, 18.723, -76.197]
  MoveL 11146 to (219.93, 34.93, 153.89) mm, rotated rx 180 ry 0 rz 180 deg; joints [-18.219, 2.648, 82.959, 76.902, 18.723, -76.197]
  Call Extruder(195.20742)
  MoveL 11147 to (221.1, 34.98, 153.89) mm, rotated rx 180 ry 0 rz -180 deg; joints [-18.181, 2.827, 82.773, 76.851, 18.688, -76.147]
  MoveL 11148 to (221.1, 34.98, 153.89) mm, rotated rx 180 ry 0 rz -180 deg; joints [-18.181, 2.827, 82.773, 76.851, 18.688, -76.147]
  Call Extruder(195.64158)
  MoveL 11149 to (221.97, 35.02, 153.89) mm, rotated rx 180 ry 0 rz 180 deg; joints [-18.154, 2.962, 82.632, 76.813, 18.664, -76.109]
  MoveL 11150 to (221.97, 35.02, 153.89) mm, rotated rx 180 ry 0 rz 180 deg; joints [-18.154, 2.962, 82.632, 76.813, 18.664, -76.109]
  Call Extruder(195.93548)
  MoveL 11151 to (222.56, 35.07, 153.89) mm, rotated rx 180 ry 0 rz -180 deg; joints [-18.138, 3.054, 82.536, 76.788, 18.649, -76.084]
  MoveL 11152 to (222.56, 35.07, 153.89) mm, rotated rx 180 ry 0 rz -180 deg; joints [-18.138, 3.054, 82.536, 76.788, 18.649, -76.084]
  Call Extruder(196.23072)
  MoveL 11153 to (223.15, 35.12, 153.89) mm, rotated rx 180 ry 0 rz 180 deg; joints [-18.122, 3.145, 82.439, 76.763, 18.634, -76.058]
  MoveL 11154 to (223.15, 35.12, 153.89) mm, rotated rx 180 ry 0 rz 180 deg; joints [-18.122, 3.145, 82.439, 76.763, 18.634, -76.058]
  Call Extruder(196.47684)
  MoveL 11155 to (223.64, 35.16, 153.89) mm, rotated rx 180 ry 0 rz 180 deg; joints [-18.109, 3.222, 82.359, 76.742, 18.623, -76.037]
  MoveL 11156 to (223.64, 35.16, 153.89) mm, rotated rx 180 ry 0 rz 180 deg; joints [-18.109, 3.222, 82.359, 76.742, 18.623, -76.037]
  Call Extruder(196.67350)
  MoveL 11157 to (224.03, 35.21, 153.89) mm, rotated rx -180 ry 0 rz 180 deg; joints [-18.1, 3.283, 82.294, 76.726, 18.615, -76.021]
  MoveL 11158 to (224.03, 35.21, 153.89) mm, rotated rx -180 ry 0 rz 180 deg; joints [-18.1, 3.283, 82.294, 76.726, 18.615, -76.021]
  Call Extruder(196.87102)
  MoveL 11159 to (224.42, 35.25, 153.89) mm, rotated rx -180 ry 0 rz -180 deg; joints [-18.091, 3.345, 82.23, 76.71, 18.607, -76.005]
  MoveL 11160 to (224.42, 35.25, 153.89) mm, rotated rx -180 ry 0 rz -180 deg; joints [-18.091, 3.345, 82.23, 76.71, 18.607, -76.005]
  Call Extruder(197.06941)
  MoveL 11161 to (224.8, 35.3, 153.89) mm, rotated rx 180 ry 0 rz 180 deg; joints [-18.083, 3.406, 82.165, 76.694, 18.599, -75.988]
  MoveL 11162 to (224.8, 35.3, 153.89) mm, rotated rx 180 ry 0 rz 180 deg; joints [-18.083, 3.406, 82.165, 76.694, 18.599, -75.988]
  Call Extruder(197.26866)
  MoveL 11163 to (225.19, 35.35, 153.89) mm, rotated rx 180 ry 0 rz 180 deg; joints [-18.074, 3.467, 82.101, 76.677, 18.592, -75.972]
  MoveL 11164 to (225.19, 35.35, 153.89) mm, rotated rx 180 ry 0 rz 180 deg; joints [-18.074, 3.467, 82.101, 76.677, 18.592, -75.972]
  Call Extruder(197.42740)
  MoveL 11165 to (225.5, 35.4, 153.89) mm, rotated rx 180 ry 0 rz 180 deg; joints [-18.068, 3.516, 82.049, 76.665, 18.587, -75.959]
  MoveL 11166 to (225.5, 35.4, 153.89) mm, rotated rx 180 ry 0 rz 180 deg; joints [-18.068, 3.516, 82.049, 76.665, 18.587, -75.959]
  Call Extruder(197.58687)
  MoveL 11167 to (225.8, 35.44, 153.89) mm, rotated rx -180 ry 0 rz 180 deg; joints [-18.062, 3.565, 81.997, 76.652, 18.582, -75.947]
  MoveL 11168 to (225.8, 35.44, 153.89) mm, rotated rx -180 ry 0 rz 180 deg; joints [-18.062, 3.565, 81.997, 76.652, 18.582, -75.947]
  Call Extruder(197.74706)
  MoveL 11169 to (226.11, 35.49, 153.89) mm, rotated rx 180 ry 0 rz 180 deg; joints [-18.057, 3.614, 81.945, 76.64, 18.577, -75.934]
  MoveL 11170 to (226.11, 35.49, 153.89) mm, rotated rx 180 ry 0 rz 180 deg; joints [-18.057, 3.614, 81.945, 76.64, 18.577, -75.934]
  Call Extruder(197.90798)
  MoveL 11171 to (226.41, 35.54, 153.89) mm, rotated rx 180 ry 0 rz 180 deg; joints [-18.051, 3.663, 81.893, 76.627, 18.572, -75.921]
  MoveL 11172 to (226.41, 35.54, 153.89) mm, rotated rx 180 ry 0 rz 180 deg; joints [-18.051, 3.663, 81.893, 76.627, 18.572, -75.921]
  Call Extruder(198.06962)
  MoveL 11173 to (226.72, 35.59, 153.89) mm, rotated rx 180 ry 0 rz -180 deg; joints [-18.045, 3.712, 81.841, 76.615, 18.567, -75.908]
  MoveL 11174 to (226.72, 35.59, 153.89) mm, rotated rx 180 ry 0 rz -180 deg; joints [-18.045, 3.712, 81.841, 76.615, 18.567, -75.908]
  Call Extruder(198.23200)
  MoveL 11175 to (227.02, 35.64, 153.89) mm, rotated rx 180 ry 0 rz 180 deg; joints [-18.04, 3.761, 81.79, 76.602, 18.563, -75.895]
  MoveL 11176 to (227.02, 35.64, 153.89) mm, rotated rx 180 ry 0 rz 180 deg; joints [-18.04, 3.761, 81.79, 76.602, 18.563, -75.895]
  Call Extruder(198.36589)
  MoveL 11177 to (227.27, 35.69, 153.89) mm, rotated rx -180 ry 0 rz 180 deg; joints [-18.036, 3.802, 81.747, 76.592, 18.56, -75.885]
  MoveL 11178 to (227.27, 35.69, 153.89) mm, rotated rx -180 ry 0 rz 180 deg; joints [-18.036, 3.802, 81.747, 76.592, 18.56, -75.885]
  Call Extruder(198.50039)
  MoveL 11179 to (227.52, 35.74, 153.89) mm, rotated rx 180 ry 0 rz 180 deg; joints [-18.033, 3.842, 81.703, 76.582, 18.557, -75.875]
  MoveL 11180 to (227.52, 35.74, 153.89) mm, rotated rx 180 ry 0 rz 180 deg; joints [-18.033, 3.842, 81.703, 76.582, 18.557, -75.875]
  Call Extruder(198.63550)
  MoveL 11181 to (227.77, 35.79, 153.89) mm, rotated rx 180 ry 0 rz 180 deg; joints [-18.029, 3.883, 81.66, 76.572, 18.554, -75.865]
  MoveL 11182 to (227.77, 35.79, 153.89) mm, rotated rx 180 ry 0 rz 180 deg; joints [-18.029, 3.883, 81.66, 76.572, 18.554, -75.865]
  Call Extruder(198.77122)
  MoveL 11183 to (228.02, 35.84, 153.89) mm, rotated rx 180 ry 0 rz 180 deg; joints [-18.026, 3.923, 81.617, 76.562, 18.552, -75.855]
  MoveL 11184 to (228.02, 35.84, 153.89) mm, rotated rx 180 ry 0 rz 180 deg; joints [-18.026, 3.923, 81.617, 76.562, 18.552, -75.855]
  Call Extruder(198.90755)
  MoveL 11185 to (228.27, 35.89, 153.89) mm, rotated rx 180 ry 0 rz 180 deg; joints [-18.022, 3.964, 81.574, 76.552, 18.549, -75.844]
  MoveL 11186 to (228.27, 35.89, 153.89) mm, rotated rx 180 ry 0 rz 180 deg; joints [-18.022, 3.964, 81.574, 76.552, 18.549, -75.844]
  Call Extruder(199.04449)
  MoveL 11187 to (228.52, 35.94, 153.89) mm, rotated rx -180 ry 0 rz 180 deg; joints [-18.019, 4.004, 81.531, 76.542, 18.546, -75.834]
  MoveL 11188 to (228.52, 35.94, 153.89) mm, rotated rx -180 ry 0 rz 180 deg; joints [-18.019, 4.004, 81.531, 76.542, 18.546, -75.834]
  Call Extruder(199.18204)
  MoveL 11189 to (228.77, 35.98, 153.89) mm, rotated rx 180 ry 0 rz -180 deg; joints [-18.016, 4.045, 81.488, 76.532, 18.543, -75.823]
  MoveL 11190 to (228.77, 35.98, 153.89) mm, rotated rx 180 ry 0 rz -180 deg; joints [-18.016, 4.045, 81.488, 76.532, 18.543, -75.823]
  Call Extruder(199.30492)
  MoveL 11191 to (228.99, 36.03, 153.89) mm, rotated rx 180 ry 0 rz -180 deg; joints [-18.013, 4.081, 81.449, 76.523, 18.541, -75.814]
  MoveL 11192 to (228.99, 36.03, 153.89) mm, rotated rx 180 ry 0 rz -180 deg; joints [-18.013, 4.081, 81.449, 76.523, 18.541, -75.814]
  Call Extruder(199.42833)
  MoveL 11193 to (229.21, 36.08, 153.89) mm, rotated rx 180 ry 0 rz 180 deg; joints [-18.011, 4.117, 81.411, 76.514, 18.54, -75.805]
  MoveL 11194 to (229.21, 36.08, 153.89) mm, rotated rx 180 ry 0 rz 180 deg; joints [-18.011, 4.117, 81.411, 76.514, 18.54, -75.805]
  Call Extruder(199.55228)
  MoveL 11195 to (229.43, 36.13, 153.89) mm, rotated rx -180 ry 0 rz -180 deg; joints [-18.008, 4.153, 81.372, 76.505, 18.538, -75.796]
  MoveL 11196 to (229.43, 36.13, 153.89) mm, rotated rx -180 ry 0 rz -180 deg; joints [-18.008, 4.153, 81.372, 76.505, 18.538, -75.796]
  Call Extruder(199.67675)
  MoveL 11197 to (229.65, 36.18, 153.89) mm, rotated rx -180 ry 0 rz -180 deg; joints [-18.005, 4.19, 81.334, 76.496, 18.536, -75.787]
  MoveL 11198 to (229.65, 36.18, 153.89) mm, rotated rx -180 ry 0 rz -180 deg; joints [-18.005, 4.19, 81.334, 76.496, 18.536, -75.787]
  Call Extruder(199.79915)
  MoveL 11199 to (229.87, 36.24, 153.89) mm, rotated rx 180 ry 0 rz 180 deg; joints [-18.004, 4.225, 81.296, 76.488, 18.535, -75.778]
  MoveL 11200 to (229.87, 36.24, 153.89) mm, rotated rx 180 ry 0 rz 180 deg; joints [-18.004, 4.225, 81.296, 76.488, 18.535, -75.778]
  Call Extruder(199.91963)
  MoveL 11201 to (230.07, 36.3, 153.89) mm, rotated rx -180 ry 0 rz 180 deg; joints [-18.004, 4.26, 81.258, 76.481, 18.535, -75.771]
  MoveL 11202 to (230.07, 36.3, 153.89) mm, rotated rx -180 ry 0 rz 180 deg; joints [-18.004, 4.26, 81.258, 76.481, 18.535, -75.771]
  Call Extruder(200.04059)
  MoveL 11203 to (230.28, 36.36, 153.89) mm, rotated rx 180 ry 0 rz 180 deg; joints [-18.003, 4.295, 81.221, 76.474, 18.535, -75.763]
  MoveL 11204 to (230.28, 36.36, 153.89) mm, rotated rx 180 ry 0 rz 180 deg; joints [-18.003, 4.295, 81.221, 76.474, 18.535, -75.763]
  Call Extruder(200.16205)
  MoveL 11205 to (230.49, 36.42, 153.89) mm, rotated rx -180 ry 0 rz 180 deg; joints [-18.003, 4.33, 81.184, 76.466, 18.535, -75.755]
  MoveL 11206 to (230.49, 36.42, 153.89) mm, rotated rx -180 ry 0 rz 180 deg; joints [-18.003, 4.33, 81.184, 76.466, 18.535, -75.755]
  Call Extruder(200.28400)
  MoveL 11207 to (230.69, 36.49, 153.89) mm, rotated rx 180 ry 0 rz 180 deg; joints [-18.002, 4.365, 81.146, 76.459, 18.535, -75.747]
  MoveL 11208 to (230.69, 36.49, 153.89) mm, rotated rx 180 ry 0 rz 180 deg; joints [-18.002, 4.365, 81.146, 76.459, 18.535, -75.747]
  Call Extruder(200.39590)
  MoveL 11209 to (230.88, 36.55, 153.89) mm, rotated rx 180 ry 0 rz 180 deg; joints [-18.002, 4.397, 81.112, 76.452, 18.536, -75.74]
  MoveL 11210 to (230.88, 36.55, 153.89) mm, rotated rx 180 ry 0 rz 180 deg; joints [-18.002, 4.397, 81.112, 76.452, 18.536, -75.74]
  Call Extruder(200.50825)
  MoveL 11211 to (231.07, 36.61, 153.89) mm, rotated rx -180 ry 0 rz 180 deg; joints [-18.002, 4.429, 81.078, 76.446, 18.536, -75.734]
  MoveL 11212 to (231.07, 36.61, 153.89) mm, rotated rx -180 ry 0 rz 180 deg; joints [-18.002, 4.429, 81.078, 76.446, 18.536, -75.734]
  Call Extruder(200.62104)
  MoveL 11213 to (231.26, 36.67, 153.89) mm, rotated rx 180 ry 0 rz -180 deg; joints [-18.002, 4.461, 81.044, 76.439, 18.537, -75.727]
  MoveL 11214 to (231.26, 36.67, 153.89) mm, rotated rx 180 ry 0 rz -180 deg; joints [-18.002, 4.461, 81.044, 76.439, 18.537, -75.727]
  Call Extruder(200.73427)
  MoveL 11215 to (231.45, 36.73, 153.89) mm, rotated rx -180 ry 0 rz 180 deg; joints [-18.002, 4.493, 81.009, 76.432, 18.537, -75.72]
  MoveL 11216 to (231.45, 36.73, 153.89) mm, rotated rx -180 ry 0 rz 180 deg; joints [-18.002, 4.493, 81.009, 76.432, 18.537, -75.72]
  Call Extruder(200.84795)
  MoveL 11217 to (231.64, 36.79, 153.89) mm, rotated rx 180 ry 0 rz 180 deg; joints [-18.002, 4.525, 80.975, 76.426, 18.538, -75.712]
  MoveL 11218 to (231.64, 36.79, 153.89) mm, rotated rx 180 ry 0 rz 180 deg; joints [-18.002, 4.525, 80.975, 76.426, 18.538, -75.712]
  Call Extruder(201.02990)
  MoveL 11219 to (231.93, 36.91, 153.89) mm, rotated rx 180 ry 0 rz 180 deg; joints [-18.005, 4.575, 80.921, 76.417, 18.542, -75.703]
  MoveL 11220 to (231.93, 36.91, 153.89) mm, rotated rx 180 ry 0 rz 180 deg; joints [-18.005, 4.575, 80.921, 76.417, 18.542, -75.703]
  Call Extruder(201.21262)
  MoveL 11221 to (232.22, 37.04, 153.89) mm, rotated rx 180 ry 0 rz -180 deg; joints [-18.008, 4.626, 80.866, 76.408, 18.545, -75.694]
  MoveL 11222 to (232.22, 37.04, 153.89) mm, rotated rx 180 ry 0 rz -180 deg; joints [-18.008, 4.626, 80.866, 76.408, 18.545, -75.694]
  Call Extruder(201.38304)
  MoveL 11223 to (232.49, 37.15, 153.89) mm, rotated rx 180 ry 0 rz 180 deg; joints [-18.011, 4.674, 80.815, 76.4, 18.549, -75.685]
  MoveL 11224 to (232.49, 37.15, 153.89) mm, rotated rx 180 ry 0 rz 180 deg; joints [-18.011, 4.674, 80.815, 76.4, 18.549, -75.685]
  Call Extruder(201.54104)
  MoveL 11225 to (232.74, 37.26, 153.89) mm, rotated rx -180 ry 0 rz 180 deg; joints [-18.013, 4.717, 80.768, 76.393, 18.552, -75.677]
  MoveL 11226 to (232.74, 37.26, 153.89) mm, rotated rx -180 ry 0 rz 180 deg; joints [-18.013, 4.717, 80.768, 76.393, 18.552, -75.677]
  Call Extruder(201.69964)
  MoveL 11227 to (232.99, 37.36, 153.89) mm, rotated rx 180 ry 0 rz 180 deg; joints [-18.016, 4.761, 80.721, 76.386, 18.556, -75.669]
  MoveL 11228 to (232.99, 37.36, 153.89) mm, rotated rx 180 ry 0 rz 180 deg; joints [-18.016, 4.761, 80.721, 76.386, 18.556, -75.669]
  Call Extruder(201.90581)
  MoveL 11229 to (233.29, 37.54, 153.89) mm, rotated rx 180 ry 0 rz 180 deg; joints [-18.024, 4.816, 80.662, 76.38, 18.565, -75.662]
  MoveL 11230 to (233.29, 37.54, 153.89) mm, rotated rx 180 ry 0 rz 180 deg; joints [-18.024, 4.816, 80.662, 76.38, 18.565, -75.662]
  Call Extruder(202.11275)
  MoveL 11231 to (233.6, 37.71, 153.89) mm, rotated rx -180 ry 0 rz 180 deg; joints [-18.033, 4.872, 80.602, 76.374, 18.574, -75.655]
  MoveL 11232 to (233.6, 37.71, 153.89) mm, rotated rx -180 ry 0 rz 180 deg; joints [-18.033, 4.872, 80.602, 76.374, 18.574, -75.655]
  Call Extruder(202.32048)
  MoveL 11233 to (233.9, 37.89, 153.89) mm, rotated rx 180 ry 0 rz 180 deg; joints [-18.041, 4.928, 80.542, 76.368, 18.583, -75.648]
  MoveL 11234 to (233.9, 37.89, 153.89) mm, rotated rx 180 ry 0 rz 180 deg; joints [-18.041, 4.928, 80.542, 76.368, 18.583, -75.648]
  Call Extruder(202.52898)
  MoveL 11235 to (234.21, 38.07, 153.89) mm, rotated rx 180 ry 0 rz -180 deg; joints [-18.049, 4.983, 80.482, 76.361, 18.592, -75.641]
  MoveL 11236 to (234.21, 38.07, 153.89) mm, rotated rx 180 ry 0 rz -180 deg; joints [-18.049, 4.983, 80.482, 76.361, 18.592, -75.641]
  Call Extruder(202.70852)
  MoveL 11237 to (234.45, 38.24, 153.89) mm, rotated rx -180 ry 0 rz -180 deg; joints [-18.06, 5.03, 80.431, 76.359, 18.603, -75.637]
  MoveL 11238 to (234.45, 38.24, 153.89) mm, rotated rx -180 ry 0 rz -180 deg; joints [-18.06, 5.03, 80.431, 76.359, 18.603, -75.637]
  Call Extruder(203.04194)
  MoveL 11239 to (234.9, 38.57, 153.89) mm, rotated rx 180 ry 0 rz 180 deg; joints [-18.079, 5.116, 80.339, 76.354, 18.624, -75.63]
  MoveL 11240 to (234.9, 38.57, 153.89) mm, rotated rx 180 ry 0 rz 180 deg; joints [-18.079, 5.116, 80.339, 76.354, 18.624, -75.63]
  Call Extruder(203.37654)
  MoveL 11241 to (235.35, 38.9, 153.89) mm, rotated rx 180 ry 0 rz 180 deg; joints [-18.099, 5.202, 80.245, 76.348, 18.644, -75.623]
  Call Extruder(204.20449)
  MoveL 11242 to (236.39, 39.81, 153.89) mm, rotated rx 180 ry 0 rz 180 deg; joints [-18.16, 5.408, 80.022, 76.346, 18.708, -75.615]
  Call Extruder(205.03243)
  MoveL 11243 to (237.3, 40.85, 153.89) mm, rotated rx -180 ry 0 rz 180 deg; joints [-18.24, 5.601, 79.811, 76.358, 18.789, -75.621]
  Call Extruder(205.19712)
  MoveL 11244 to (237.47, 41.07, 153.89) mm, rotated rx 180 ry 0 rz -180 deg; joints [-18.258, 5.638, 79.772, 76.363, 18.807, -75.624]
  MoveL 11245 to (237.47, 41.07, 153.89) mm, rotated rx 180 ry 0 rz -180 deg; joints [-18.258, 5.638, 79.772, 76.363, 18.807, -75.624]
  Call Extruder(205.52536)
  MoveL 11246 to (237.79, 41.51, 153.89) mm, rotated rx 180 ry 0 rz -180 deg; joints [-18.294, 5.71, 79.692, 76.372, 18.844, -75.631]
  MoveL 11247 to (237.79, 41.51, 153.89) mm, rotated rx 180 ry 0 rz -180 deg; joints [-18.294, 5.71, 79.692, 76.372, 18.844, -75.631]
  Call Extruder(205.85246)
  MoveL 11248 to (238.11, 41.96, 153.89) mm, rotated rx -180 ry 0 rz -180 deg; joints [-18.33, 5.783, 79.613, 76.38, 18.88, -75.637]
  MoveL 11249 to (238.11, 41.96, 153.89) mm, rotated rx -180 ry 0 rz -180 deg; joints [-18.33, 5.783, 79.613, 76.38, 18.88, -75.637]
  Call Extruder(205.98700)
  MoveL 11250 to (238.23, 42.15, 153.89) mm, rotated rx 180 ry 0 rz -180 deg; joints [-18.347, 5.81, 79.583, 76.386, 18.897, -75.642]
  MoveL 11251 to (238.23, 42.15, 153.89) mm, rotated rx 180 ry 0 rz -180 deg; joints [-18.347, 5.81, 79.583, 76.386, 18.897, -75.642]
  Call Extruder(206.20232)
  MoveL 11252 to (238.41, 42.47, 153.89) mm, rotated rx 180 ry 0 rz 180 deg; joints [-18.374, 5.855, 79.534, 76.395, 18.925, -75.649]
  MoveL 11253 to (238.41, 42.47, 153.89) mm, rotated rx 180 ry 0 rz 180 deg; joints [-18.374, 5.855, 79.534, 76.395, 18.925, -75.649]
  Call Extruder(206.41679)
  MoveL 11254 to (238.59, 42.79, 153.89) mm, rotated rx 180 ry 0 rz 180 deg; joints [-18.402, 5.899, 79.486, 76.404, 18.952, -75.656]
  MoveL 11255 to (238.59, 42.79, 153.89) mm, rotated rx 180 ry 0 rz 180 deg; joints [-18.402, 5.899, 79.486, 76.404, 18.952, -75.656]
  Call Extruder(206.63041)
  MoveL 11256 to (238.77, 43.1, 153.89) mm, rotated rx -180 ry 0 rz 180 deg; joints [-18.429, 5.943, 79.438, 76.413, 18.98, -75.663]
  MoveL 11257 to (238.77, 43.1, 153.89) mm, rotated rx -180 ry 0 rz 180 deg; joints [-18.429, 5.943, 79.438, 76.413, 18.98, -75.663]
  Call Extruder(206.80964)
  MoveL 11258 to (238.91, 43.37, 153.89) mm, rotated rx -180 ry 0 rz -180 deg; joints [-18.453, 5.979, 79.398, 76.422, 19.004, -75.67]
  MoveL 11259 to (238.91, 43.37, 153.89) mm, rotated rx -180 ry 0 rz -180 deg; joints [-18.453, 5.979, 79.398, 76.422, 19.004, -75.67]
  Call Extruder(206.95538)
  MoveL 11260 to (239.01, 43.6, 153.89) mm, rotated rx 180 ry 0 rz 180 deg; joints [-18.474, 6.006, 79.369, 76.43, 19.025, -75.678]
  MoveL 11261 to (239.01, 43.6, 153.89) mm, rotated rx 180 ry 0 rz 180 deg; joints [-18.474, 6.006, 79.369, 76.43, 19.025, -75.678]
  Call Extruder(207.10061)
  MoveL 11262 to (239.11, 43.83, 153.89) mm, rotated rx 180 ry 0 rz 180 deg; joints [-18.495, 6.033, 79.339, 76.439, 19.046, -75.685]
  MoveL 11263 to (239.11, 43.83, 153.89) mm, rotated rx 180 ry 0 rz 180 deg; joints [-18.495, 6.033, 79.339, 76.439, 19.046, -75.685]
  Call Extruder(207.28332)
  MoveL 11264 to (239.22, 44.13, 153.89) mm, rotated rx 180 ry 0 rz -180 deg; joints [-18.522, 6.067, 79.302, 76.45, 19.072, -75.694]
  MoveL 11265 to (239.22, 44.13, 153.89) mm, rotated rx 180 ry 0 rz -180 deg; joints [-18.522, 6.067, 79.302, 76.45, 19.072, -75.694]
  Call Extruder(207.46527)
  MoveL 11266 to (239.35, 44.42, 153.89) mm, rotated rx -180 ry 0 rz -180 deg; joints [-18.549, 6.101, 79.265, 76.461, 19.099, -75.704]
  MoveL 11267 to (239.35, 44.42, 153.89) mm, rotated rx -180 ry 0 rz -180 deg; joints [-18.549, 6.101, 79.265, 76.461, 19.099, -75.704]
  Call Extruder(207.61260)
  MoveL 11268 to (239.44, 44.66, 153.89) mm, rotated rx -180 ry 0 rz -180 deg; joints [-18.571, 6.127, 79.236, 76.47, 19.121, -75.712]
  MoveL 11269 to (239.44, 44.66, 153.89) mm, rotated rx -180 ry 0 rz -180 deg; joints [-18.571, 6.127, 79.236, 76.47, 19.121, -75.712]
  Call Extruder(207.72584)
  MoveL 11270 to (239.5, 44.85, 153.89) mm, rotated rx -180 ry 0 rz -180 deg; joints [-18.589, 6.147, 79.214, 76.479, 19.139, -75.719]
  MoveL 11271 to (239.5, 44.85, 153.89) mm, rotated rx -180 ry 0 rz -180 deg; joints [-18.589, 6.147, 79.214, 76.479, 19.139, -75.719]
  Call Extruder(207.83863)
  MoveL 11272 to (239.56, 45.03, 153.89) mm, rotated rx 180 ry 0 rz 180 deg; joints [-18.607, 6.166, 79.193, 76.487, 19.157, -75.726]
  MoveL 11273 to (239.56, 45.03, 153.89) mm, rotated rx 180 ry 0 rz 180 deg; joints [-18.607, 6.166, 79.193, 76.487, 19.157, -75.726]
  Call Extruder(207.95098)
  MoveL 11274 to (239.62, 45.22, 153.89) mm, rotated rx -180 ry 0 rz -180 deg; joints [-18.625, 6.185, 79.172, 76.495, 19.175, -75.733]
  MoveL 11275 to (239.62, 45.22, 153.89) mm, rotated rx -180 ry 0 rz -180 deg; joints [-18.625, 6.185, 79.172, 76.495, 19.175, -75.733]
  Call Extruder(208.06288)
  MoveL 11276 to (239.68, 45.41, 153.89) mm, rotated rx -180 ry 0 rz 180 deg; joints [-18.642, 6.205, 79.151, 76.503, 19.192, -75.74]
  MoveL 11277 to (239.68, 45.41, 153.89) mm, rotated rx -180 ry 0 rz 180 deg; joints [-18.642, 6.205, 79.151, 76.503, 19.192, -75.74]
  Call Extruder(208.18428)
  MoveL 11278 to (239.75, 45.62, 153.89) mm, rotated rx 180 ry 0 rz 180 deg; joints [-18.662, 6.225, 79.128, 76.512, 19.212, -75.748]
  MoveL 11279 to (239.75, 45.62, 153.89) mm, rotated rx 180 ry 0 rz 180 deg; joints [-18.662, 6.225, 79.128, 76.512, 19.212, -75.748]
  Call Extruder(208.31507)
  MoveL 11280 to (239.82, 45.84, 153.89) mm, rotated rx -180 ry 0 rz 180 deg; joints [-18.683, 6.248, 79.103, 76.521, 19.233, -75.756]
  MoveL 11281 to (239.82, 45.84, 153.89) mm, rotated rx -180 ry 0 rz 180 deg; joints [-18.683, 6.248, 79.103, 76.521, 19.233, -75.756]
  Call Extruder(208.44530)
  MoveL 11282 to (239.88, 46.06, 153.89) mm, rotated rx 180 ry 0 rz -180 deg; joints [-18.705, 6.27, 79.079, 76.531, 19.254, -75.765]
  MoveL 11283 to (239.88, 46.06, 153.89) mm, rotated rx 180 ry 0 rz -180 deg; joints [-18.705, 6.27, 79.079, 76.531, 19.254, -75.765]
  Call Extruder(208.57496)
  MoveL 11284 to (239.95, 46.29, 153.89) mm, rotated rx -180 ry 0 rz 180 deg; joints [-18.726, 6.292, 79.055, 76.541, 19.275, -75.773]
  MoveL 11285 to (239.95, 46.29, 153.89) mm, rotated rx -180 ry 0 rz 180 deg; joints [-18.726, 6.292, 79.055, 76.541, 19.275, -75.773]
  Call Extruder(208.70405)
  MoveL 11286 to (240.02, 46.51, 153.89) mm, rotated rx 180 ry 0 rz 180 deg; joints [-18.747, 6.314, 79.03, 76.55, 19.297, -75.781]
  MoveL 11287 to (240.02, 46.51, 153.89) mm, rotated rx 180 ry 0 rz 180 deg; joints [-18.747, 6.314, 79.03, 76.55, 19.297, -75.781]
  Call Extruder(208.81911)
  MoveL 11288 to (240.06, 46.72, 153.89) mm, rotated rx 180 ry 0 rz 180 deg; joints [-18.767, 6.332, 79.011, 76.56, 19.316, -75.79]
  MoveL 11289 to (240.06, 46.72, 153.89) mm, rotated rx 180 ry 0 rz 180 deg; joints [-18.767, 6.332, 79.011, 76.56, 19.316, -75.79]
  Call Extruder(208.93371)
  MoveL 11290 to (240.11, 46.92, 153.89) mm, rotated rx 180 ry 0 rz -180 deg; joints [-18.787, 6.349, 78.991, 76.57, 19.336, -75.799]
  MoveL 11291 to (240.11, 46.92, 153.89) mm, rotated rx 180 ry 0 rz -180 deg; joints [-18.787, 6.349, 78.991, 76.57, 19.336, -75.799]
  Call Extruder(209.04786)
  MoveL 11292 to (240.15, 47.12, 153.89) mm, rotated rx 180 ry 0 rz 180 deg; joints [-18.807, 6.367, 78.972, 76.58, 19.356, -75.808]
  MoveL 11293 to (240.15, 47.12, 153.89) mm, rotated rx 180 ry 0 rz 180 deg; joints [-18.807, 6.367, 78.972, 76.58, 19.356, -75.808]
  Call Extruder(209.16155)
  MoveL 11294 to (240.2, 47.33, 153.89) mm, rotated rx 180 ry 0 rz 180 deg; joints [-18.827, 6.385, 78.952, 76.59, 19.376, -75.816]
  MoveL 11295 to (240.2, 47.33, 153.89) mm, rotated rx 180 ry 0 rz 180 deg; joints [-18.827, 6.385, 78.952, 76.59, 19.376, -75.816]
  Call Extruder(209.28696)
  MoveL 11296 to (240.24, 47.55, 153.89) mm, rotated rx 180 ry 0 rz 180 deg; joints [-18.85, 6.404, 78.931, 76.601, 19.398, -75.826]
  MoveL 11297 to (240.24, 47.55, 153.89) mm, rotated rx 180 ry 0 rz 180 deg; joints [-18.85, 6.404, 78.931, 76.601, 19.398, -75.826]
  Call Extruder(209.42394)
  MoveL 11298 to (240.29, 47.8, 153.89) mm, rotated rx -180 ry 0 rz -180 deg; joints [-18.874, 6.425, 78.908, 76.613, 19.422, -75.837]
  MoveL 11299 to (240.29, 47.8, 153.89) mm, rotated rx -180 ry 0 rz -180 deg; joints [-18.874, 6.425, 78.908, 76.613, 19.422, -75.837]
  Call Extruder(209.56031)
  MoveL 11300 to (240.34, 48.05, 153.89) mm, rotated rx 180 ry 0 rz 180 deg; joints [-18.899, 6.446, 78.885, 76.625, 19.447, -75.847]
  MoveL 11301 to (240.34, 48.05, 153.89) mm, rotated rx 180 ry 0 rz 180 deg; joints [-18.899, 6.446, 78.885, 76.625, 19.447, -75.847]
  Call Extruder(209.69607)
  MoveL 11302 to (240.39, 48.3, 153.89) mm, rotated rx 180 ry 0 rz 180 deg; joints [-18.923, 6.467, 78.862, 76.637, 19.471, -75.858]
  MoveL 11303 to (240.39, 48.3, 153.89) mm, rotated rx 180 ry 0 rz 180 deg; joints [-18.923, 6.467, 78.862, 76.637, 19.471, -75.858]
  Call Extruder(209.83121)
  MoveL 11304 to (240.44, 48.55, 153.89) mm, rotated rx 180 ry 0 rz 180 deg; joints [-18.948, 6.488, 78.839, 76.649, 19.495, -75.869]
  MoveL 11305 to (240.44, 48.55, 153.89) mm, rotated rx 180 ry 0 rz 180 deg; joints [-18.948, 6.488, 78.839, 76.649, 19.495, -75.869]
  Call Extruder(209.96575)
  MoveL 11306 to (240.49, 48.8, 153.89) mm, rotated rx 180 ry 0 rz -180 deg; joints [-18.973, 6.509, 78.816, 76.661, 19.52, -75.879]
  MoveL 11307 to (240.49, 48.8, 153.89) mm, rotated rx 180 ry 0 rz -180 deg; joints [-18.973, 6.509, 78.816, 76.661, 19.52, -75.879]
  Call Extruder(210.09968)
  MoveL 11308 to (240.54, 49.05, 153.89) mm, rotated rx 180 ry 0 rz -180 deg; joints [-18.997, 6.529, 78.793, 76.673, 19.544, -75.89]
  MoveL 11309 to (240.54, 49.05, 153.89) mm, rotated rx 180 ry 0 rz -180 deg; joints [-18.997, 6.529, 78.793, 76.673, 19.544, -75.89]
  Call Extruder(210.24754)
  MoveL 11310 to (240.59, 49.33, 153.89) mm, rotated rx -180 ry 0 rz 180 deg; joints [-19.025, 6.552, 78.768, 76.686, 19.571, -75.902]
  MoveL 11311 to (240.59, 49.33, 153.89) mm, rotated rx -180 ry 0 rz 180 deg; joints [-19.025, 6.552, 78.768, 76.686, 19.571, -75.902]
  Call Extruder(210.40929)
  MoveL 11312 to (240.64, 49.63, 153.89) mm, rotated rx 180 ry 0 rz 180 deg; joints [-19.055, 6.576, 78.742, 76.702, 19.601, -75.915]
  MoveL 11313 to (240.64, 49.63, 153.89) mm, rotated rx 180 ry 0 rz 180 deg; joints [-19.055, 6.576, 78.742, 76.702, 19.601, -75.915]
  Call Extruder(210.57031)
  MoveL 11314 to (240.69, 49.94, 153.89) mm, rotated rx 180 ry 0 rz 180 deg; joints [-19.086, 6.6, 78.715, 76.717, 19.631, -75.929]
  MoveL 11315 to (240.69, 49.94, 153.89) mm, rotated rx 180 ry 0 rz 180 deg; joints [-19.086, 6.6, 78.715, 76.717, 19.631, -75.929]
  Call Extruder(210.73060)
  MoveL 11316 to (240.74, 50.24, 153.89) mm, rotated rx 180 ry 0 rz 180 deg; joints [-19.116, 6.624, 78.689, 76.732, 19.662, -75.942]
  MoveL 11317 to (240.74, 50.24, 153.89) mm, rotated rx 180 ry 0 rz 180 deg; joints [-19.116, 6.624, 78.689, 76.732, 19.662, -75.942]
  Call Extruder(210.89016)
  MoveL 11318 to (240.78, 50.55, 153.89) mm, rotated rx 180 ry 0 rz 180 deg; joints [-19.146, 6.647, 78.662, 76.747, 19.692, -75.956]
  MoveL 11319 to (240.78, 50.55, 153.89) mm, rotated rx 180 ry 0 rz 180 deg; joints [-19.146, 6.647, 78.662, 76.747, 19.692, -75.956]
  Call Extruder(211.04899)
  MoveL 11320 to (240.83, 50.86, 153.89) mm, rotated rx -180 ry 0 rz 180 deg; joints [-19.177, 6.671, 78.636, 76.762, 19.722, -75.969]
  MoveL 11321 to (240.83, 50.86, 153.89) mm, rotated rx -180 ry 0 rz 180 deg; joints [-19.177, 6.671, 78.636, 76.762, 19.722, -75.969]
  Call Extruder(211.22766)
  MoveL 11322 to (240.88, 51.2, 153.89) mm, rotated rx -180 ry 0 rz 180 deg; joints [-19.212, 6.697, 78.607, 76.779, 19.756, -75.984]
  MoveL 11323 to (240.88, 51.2, 153.89) mm, rotated rx -180 ry 0 rz 180 deg; joints [-19.212, 6.697, 78.607, 76.779, 19.756, -75.984]
  Call Extruder(211.42611)
  MoveL 11324 to (240.92, 51.59, 153.89) mm, rotated rx -180 ry 0 rz 180 deg; joints [-19.251, 6.725, 78.576, 76.799, 19.795, -76.002]
  MoveL 11325 to (240.92, 51.59, 153.89) mm, rotated rx -180 ry 0 rz 180 deg; joints [-19.251, 6.725, 78.576, 76.799, 19.795, -76.002]
  Call Extruder(211.62368)
  MoveL 11326 to (240.97, 51.98, 153.89) mm, rotated rx 180 ry 0 rz -180 deg; joints [-19.29, 6.754, 78.545, 76.819, 19.833, -76.019]
  MoveL 11327 to (240.97, 51.98, 153.89) mm, rotated rx 180 ry 0 rz -180 deg; joints [-19.29, 6.754, 78.545, 76.819, 19.833, -76.019]
  Call Extruder(211.82039)
  MoveL 11328 to (241.02, 52.37, 153.89) mm, rotated rx -180 ry 0 rz 180 deg; joints [-19.329, 6.782, 78.513, 76.838, 19.872, -76.037]
  MoveL 11329 to (241.02, 52.37, 153.89) mm, rotated rx -180 ry 0 rz 180 deg; joints [-19.329, 6.782, 78.513, 76.838, 19.872, -76.037]
  Call Extruder(212.01622)
  MoveL 11330 to (241.06, 52.75, 153.89) mm, rotated rx 180 ry 0 rz 180 deg; joints [-19.368, 6.81, 78.482, 76.858, 19.911, -76.054]
  MoveL 11331 to (241.06, 52.75, 153.89) mm, rotated rx 180 ry 0 rz 180 deg; joints [-19.368, 6.81, 78.482, 76.858, 19.911, -76.054]
  Call Extruder(212.31166)
  MoveL 11332 to (241.11, 53.34, 153.89) mm, rotated rx 180 ry 0 rz -180 deg; joints [-19.428, 6.849, 78.439, 76.889, 19.97, -76.082]
  MoveL 11333 to (241.11, 53.34, 153.89) mm, rotated rx 180 ry 0 rz -180 deg; joints [-19.428, 6.849, 78.439, 76.889, 19.97, -76.082]
  Call Extruder(212.60577)
  MoveL 11334 to (241.15, 53.93, 153.89) mm, rotated rx 180 ry 0 rz 180 deg; joints [-19.488, 6.889, 78.395, 76.919, 20.029, -76.109]
  MoveL 11335 to (241.15, 53.93, 153.89) mm, rotated rx 180 ry 0 rz 180 deg; joints [-19.488, 6.889, 78.395, 76.919, 20.029, -76.109]
  Call Extruder(212.89854)
  MoveL 11336 to (241.2, 54.52, 153.89) mm, rotated rx 180 ry 0 rz 180 deg; joints [-19.548, 6.928, 78.351, 76.95, 20.089, -76.136]
  MoveL 11337 to (241.2, 54.52, 153.89) mm, rotated rx 180 ry 0 rz 180 deg; joints [-19.548, 6.928, 78.351, 76.95, 20.089, -76.136]
  Call Extruder(213.47199)
  MoveL 11338 to (241.25, 55.68, 153.89) mm, rotated rx -180 ry 0 rz 180 deg; joints [-19.668, 6.999, 78.272, 77.012, 20.207, -76.192]
  MoveL 11339 to (241.25, 55.68, 153.89) mm, rotated rx -180 ry 0 rz 180 deg; joints [-19.668, 6.999, 78.272, 77.012, 20.207, -76.192]
  Call Extruder(214.18582)
  MoveL 11340 to (241.29, 57.14, 153.89) mm, rotated rx 180 ry 0 rz -180 deg; joints [-19.819, 7.086, 78.175, 77.089, 20.355, -76.261]
  Call Extruder(256.25069)
  MoveL 11341 to (241.29, 142.86, 153.89) mm, rotated rx 180 ry 0 rz 180 deg; joints [-28.232, 13.003, 71.305, 79.535, 28.754, -78.102]
  Call Extruder(256.67912)
  MoveL 11342 to (241.27, 143.74, 153.89) mm, rotated rx 180 ry 0 rz 180 deg; joints [-28.313, 13.073, 71.221, 79.543, 28.835, -78.103]
  MoveL 11343 to (241.27, 143.74, 153.89) mm, rotated rx 180 ry 0 rz 180 deg; joints [-28.313, 13.073, 71.221, 79.543, 28.835, -78.103]
  Call Extruder(257.25257)
  MoveL 11344 to (241.22, 144.9, 153.89) mm, rotated rx -180 ry 0 rz 180 deg; joints [-28.421, 13.162, 71.113, 79.556, 28.945, -78.105]
  MoveL 11345 to (241.22, 144.9, 153.89) mm, rotated rx -180 ry 0 rz 180 deg; joints [-28.421, 13.162, 71.113, 79.556, 28.945, -78.105]
  Call Extruder(257.68690)
  MoveL 11346 to (241.18, 145.77, 153.89) mm, rotated rx 180 ry 0 rz 180 deg; joints [-28.503, 13.228, 71.033, 79.566, 29.028, -78.108]
  MoveL 11347 to (241.18, 145.77, 153.89) mm, rotated rx 180 ry 0 rz 180 deg; joints [-28.503, 13.228, 71.033, 79.566, 29.028, -78.108]
  Call Extruder(257.98101)
  MoveL 11348 to (241.13, 146.36, 153.89) mm, rotated rx 180 ry 0 rz 180 deg; joints [-28.559, 13.27, 70.982, 79.574, 29.084, -78.11]
  MoveL 11349 to (241.13, 146.36, 153.89) mm, rotated rx 180 ry 0 rz 180 deg; joints [-28.559, 13.27, 70.982, 79.574, 29.084, -78.11]
  Call Extruder(258.27645)
  MoveL 11350 to (241.09, 146.95, 153.89) mm, rotated rx 180 ry 0 rz 180 deg; joints [-28.615, 13.312, 70.931, 79.582, 29.141, -78.113]
  MoveL 11351 to (241.09, 146.95, 153.89) mm, rotated rx 180 ry 0 rz 180 deg; joints [-28.615, 13.312, 70.931, 79.582, 29.141, -78.113]
  Call Extruder(258.52270)
  MoveL 11352 to (241.04, 147.44, 153.89) mm, rotated rx -180 ry 0 rz 180 deg; joints [-28.662, 13.346, 70.89, 79.589, 29.188, -78.115]
  MoveL 11353 to (241.04, 147.44, 153.89) mm, rotated rx -180 ry 0 rz 180 deg; joints [-28.662, 13.346, 70.89, 79.589, 29.188, -78.115]
  Call Extruder(258.71941)
  MoveL 11354 to (240.99, 147.83, 153.89) mm, rotated rx 180 ry 0 rz 180 deg; joints [-28.7, 13.372, 70.859, 79.595, 29.225, -78.118]
  MoveL 11355 to (240.99, 147.83, 153.89) mm, rotated rx 180 ry 0 rz 180 deg; joints [-28.7, 13.372, 70.859, 79.595, 29.225, -78.118]
  Call Extruder(258.91698)
  MoveL 11356 to (240.95, 148.22, 153.89) mm, rotated rx -180 ry 0 rz 180 deg; joints [-28.737, 13.397, 70.828, 79.601, 29.263, -78.121]
  MoveL 11357 to (240.95, 148.22, 153.89) mm, rotated rx -180 ry 0 rz 180 deg; joints [-28.737, 13.397, 70.828, 79.601, 29.263, -78.121]
  Call Extruder(259.11542)
  MoveL 11358 to (240.9, 148.6, 153.89) mm, rotated rx 180 ry 0 rz 180 deg; joints [-28.774, 13.423, 70.797, 79.608, 29.301, -78.124]
  MoveL 11359 to (240.9, 148.6, 153.89) mm, rotated rx 180 ry 0 rz 180 deg; joints [-28.774, 13.423, 70.797, 79.608, 29.301, -78.124]
  Call Extruder(259.31473)
  MoveL 11360 to (240.86, 148.99, 153.89) mm, rotated rx 180 ry 0 rz 180 deg; joints [-28.812, 13.449, 70.765, 79.614, 29.338, -78.126]
  MoveL 11361 to (240.86, 148.99, 153.89) mm, rotated rx 180 ry 0 rz 180 deg; joints [-28.812, 13.449, 70.765, 79.614, 29.338, -78.126]
  Call Extruder(259.47356)
  MoveL 11362 to (240.81, 149.3, 153.89) mm, rotated rx 180 ry 0 rz 180 deg; joints [-28.842, 13.467, 70.743, 79.619, 29.368, -78.129]
  MoveL 11363 to (240.81, 149.3, 153.89) mm, rotated rx 180 ry 0 rz 180 deg; joints [-28.842, 13.467, 70.743, 79.619, 29.368, -78.129]
  Call Extruder(259.63312)
  MoveL 11364 to (240.76, 149.6, 153.89) mm, rotated rx 180 ry 0 rz 180 deg; joints [-28.872, 13.485, 70.721, 79.625, 29.399, -78.132]
  MoveL 11365 to (240.76, 149.6, 153.89) mm, rotated rx 180 ry 0 rz 180 deg; joints [-28.872, 13.485, 70.721, 79.625, 29.399, -78.132]
  Call Extruder(259.79341)
  MoveL 11366 to (240.71, 149.91, 153.89) mm, rotated rx -180 ry 0 rz 180 deg; joints [-28.902, 13.504, 70.698, 79.631, 29.429, -78.135]
  MoveL 11367 to (240.71, 149.91, 153.89) mm, rotated rx -180 ry 0 rz 180 deg; joints [-28.902, 13.504, 70.698, 79.631, 29.429, -78.135]
  Call Extruder(259.95443)
  MoveL 11368 to (240.66, 150.21, 153.89) mm, rotated rx -180 ry 0 rz 180 deg; joints [-28.932, 13.522, 70.676, 79.636, 29.459, -78.138]
  MoveL 11369 to (240.66, 150.21, 153.89) mm, rotated rx -180 ry 0 rz 180 deg; joints [-28.932, 13.522, 70.676, 79.636, 29.459, -78.138]
  Call Extruder(260.11618)
  MoveL 11370 to (240.61, 150.52, 153.89) mm, rotated rx 180 ry 0 rz 180 deg; joints [-28.962, 13.541, 70.653, 79.642, 29.489, -78.141]
  MoveL 11371 to (240.61, 150.52, 153.89) mm, rotated rx 180 ry 0 rz 180 deg; joints [-28.962, 13.541, 70.653, 79.642, 29.489, -78.141]
  Call Extruder(260.27865)
  MoveL 11372 to (240.57, 150.83, 153.89) mm, rotated rx -180 ry 0 rz 180 deg; joints [-28.993, 13.559, 70.631, 79.647, 29.519, -78.144]
  MoveL 11373 to (240.57, 150.83, 153.89) mm, rotated rx -180 ry 0 rz 180 deg; joints [-28.993, 13.559, 70.631, 79.647, 29.519, -78.144]
  Call Extruder(260.41257)
  MoveL 11374 to (240.52, 151.08, 153.89) mm, rotated rx 180 ry 0 rz 180 deg; joints [-29.017, 13.573, 70.614, 79.653, 29.544, -78.147]
  MoveL 11375 to (240.52, 151.08, 153.89) mm, rotated rx 180 ry 0 rz 180 deg; joints [-29.017, 13.573, 70.614, 79.653, 29.544, -78.147]
  Call Extruder(260.54711)
  MoveL 11376 to (240.47, 151.32, 153.89) mm, rotated rx 180 ry 0 rz 180 deg; joints [-29.043, 13.587, 70.597, 79.658, 29.569, -78.15]
  MoveL 11377 to (240.47, 151.32, 153.89) mm, rotated rx 180 ry 0 rz 180 deg; joints [-29.043, 13.587, 70.597, 79.658, 29.569, -78.15]
  Call Extruder(260.68226)
  MoveL 11378 to (240.42, 151.57, 153.89) mm, rotated rx 180 ry 0 rz 180 deg; joints [-29.067, 13.6, 70.581, 79.663, 29.594, -78.154]
  MoveL 11379 to (240.42, 151.57, 153.89) mm, rotated rx 180 ry 0 rz 180 deg; joints [-29.067, 13.6, 70.581, 79.663, 29.594, -78.154]
  Call Extruder(260.81801)
  MoveL 11380 to (240.37, 151.82, 153.89) mm, rotated rx 180 ry 0 rz 180 deg; joints [-29.092, 13.614, 70.564, 79.668, 29.619, -78.157]
  MoveL 11381 to (240.37, 151.82, 153.89) mm, rotated rx 180 ry 0 rz 180 deg; joints [-29.092, 13.614, 70.564, 79.668, 29.619, -78.157]
  Call Extruder(260.95438)
  MoveL 11382 to (240.32, 152.07, 153.89) mm, rotated rx 180 ry 0 rz 180 deg; joints [-29.117, 13.628, 70.548, 79.674, 29.644, -78.16]
  MoveL 11383 to (240.32, 152.07, 153.89) mm, rotated rx 180 ry 0 rz 180 deg; joints [-29.117, 13.628, 70.548, 79.674, 29.644, -78.16]
  Call Extruder(261.09136)
  MoveL 11384 to (240.27, 152.32, 153.89) mm, rotated rx 180 ry 0 rz 180 deg; joints [-29.142, 13.641, 70.531, 79.679, 29.669, -78.163]
  MoveL 11385 to (240.27, 152.32, 153.89) mm, rotated rx 180 ry 0 rz 180 deg; joints [-29.142, 13.641, 70.531, 79.679, 29.669, -78.163]
  Call Extruder(261.22895)
  MoveL 11386 to (240.22, 152.57, 153.89) mm, rotated rx 180 ry 0 rz 180 deg; joints [-29.167, 13.655, 70.514, 79.684, 29.694, -78.166]
  MoveL 11387 to (240.22, 152.57, 153.89) mm, rotated rx 180 ry 0 rz 180 deg; joints [-29.167, 13.655, 70.514, 79.684, 29.694, -78.166]
  Call Extruder(261.34265)
  MoveL 11388 to (240.17, 152.77, 153.89) mm, rotated rx -180 ry 0 rz 180 deg; joints [-29.188, 13.666, 70.501, 79.688, 29.715, -78.168]
  MoveL 11389 to (240.17, 152.77, 153.89) mm, rotated rx -180 ry 0 rz 180 deg; joints [-29.188, 13.666, 70.501, 79.688, 29.715, -78.168]
  Call Extruder(261.45680)
  MoveL 11390 to (240.13, 152.98, 153.89) mm, rotated rx -180 ry 0 rz 180 deg; joints [-29.209, 13.676, 70.488, 79.693, 29.735, -78.171]
  MoveL 11391 to (240.13, 152.98, 153.89) mm, rotated rx -180 ry 0 rz 180 deg; joints [-29.209, 13.676, 70.488, 79.693, 29.735, -78.171]
  Call Extruder(261.57140)
  MoveL 11392 to (240.08, 153.18, 153.89) mm, rotated rx -180 ry 0 rz 180 deg; joints [-29.229, 13.687, 70.475, 79.698, 29.756, -78.174]
  MoveL 11393 to (240.08, 153.18, 153.89) mm, rotated rx -180 ry 0 rz 180 deg; joints [-29.229, 13.687, 70.475, 79.698, 29.756, -78.174]
  Call Extruder(261.68645)
  MoveL 11394 to (240.04, 153.39, 153.89) mm, rotated rx 180 ry 0 rz 180 deg; joints [-29.25, 13.698, 70.462, 79.702, 29.777, -78.177]
  MoveL 11395 to (240.04, 153.39, 153.89) mm, rotated rx 180 ry 0 rz 180 deg; joints [-29.25, 13.698, 70.462, 79.702, 29.777, -78.177]
  Call Extruder(261.80867)
  MoveL 11396 to (239.98, 153.6, 153.89) mm, rotated rx 180 ry 0 rz 180 deg; joints [-29.272, 13.708, 70.45, 79.707, 29.799, -78.18]
  MoveL 11397 to (239.98, 153.6, 153.89) mm, rotated rx 180 ry 0 rz 180 deg; joints [-29.272, 13.708, 70.45, 79.707, 29.799, -78.18]
  Call Extruder(261.93833)
  MoveL 11398 to (239.92, 153.82, 153.89) mm, rotated rx -180 ry 0 rz 180 deg; joints [-29.296, 13.716, 70.439, 79.714, 29.822, -78.185]
  MoveL 11399 to (239.92, 153.82, 153.89) mm, rotated rx -180 ry 0 rz 180 deg; joints [-29.296, 13.716, 70.439, 79.714, 29.822, -78.185]
  Call Extruder(262.06856)
  MoveL 11400 to (239.85, 154.05, 153.89) mm, rotated rx 180 ry 0 rz -180 deg; joints [-29.319, 13.725, 70.429, 79.72, 29.845, -78.19]
  MoveL 11401 to (239.85, 154.05, 153.89) mm, rotated rx 180 ry 0 rz -180 deg; joints [-29.319, 13.725, 70.429, 79.72, 29.845, -78.19]
  Call Extruder(262.19935)
  MoveL 11402 to (239.78, 154.27, 153.89) mm, rotated rx 180 ry 0 rz 180 deg; joints [-29.343, 13.734, 70.418, 79.726, 29.869, -78.194]
  MoveL 11403 to (239.78, 154.27, 153.89) mm, rotated rx 180 ry 0 rz 180 deg; joints [-29.343, 13.734, 70.418, 79.726, 29.869, -78.194]
  Call Extruder(262.33071)
  MoveL 11404 to (239.71, 154.5, 153.89) mm, rotated rx 180 ry 0 rz 180 deg; joints [-29.366, 13.743, 70.407, 79.733, 29.892, -78.199]
  MoveL 11405 to (239.71, 154.5, 153.89) mm, rotated rx 180 ry 0 rz 180 deg; joints [-29.366, 13.743, 70.407, 79.733, 29.892, -78.199]
  Call Extruder(262.44261)
  MoveL 11406 to (239.65, 154.68, 153.89) mm, rotated rx 180 ry 0 rz 180 deg; joints [-29.386, 13.75, 70.398, 79.738, 29.912, -78.203]
  MoveL 11407 to (239.65, 154.68, 153.89) mm, rotated rx 180 ry 0 rz 180 deg; joints [-29.386, 13.75, 70.398, 79.738, 29.912, -78.203]
  Call Extruder(262.55495)
  MoveL 11408 to (239.59, 154.87, 153.89) mm, rotated rx 180 ry 0 rz 180 deg; joints [-29.406, 13.757, 70.39, 79.744, 29.932, -78.207]
  MoveL 11409 to (239.59, 154.87, 153.89) mm, rotated rx 180 ry 0 rz 180 deg; joints [-29.406, 13.757, 70.39, 79.744, 29.932, -78.207]
  Call Extruder(262.66774)
  MoveL 11410 to (239.53, 155.06, 153.89) mm, rotated rx 180 ry 0 rz 180 deg; joints [-29.426, 13.764, 70.382, 79.75, 29.952, -78.211]
  MoveL 11411 to (239.53, 155.06, 153.89) mm, rotated rx 180 ry 0 rz 180 deg; joints [-29.426, 13.764, 70.382, 79.75, 29.952, -78.211]
  Call Extruder(262.78098)
  MoveL 11412 to (239.47, 155.25, 153.89) mm, rotated rx 180 ry 0 rz 180 deg; joints [-29.446, 13.771, 70.373, 79.755, 29.972, -78.215]
  MoveL 11413 to (239.47, 155.25, 153.89) mm, rotated rx 180 ry 0 rz 180 deg; joints [-29.446, 13.771, 70.373, 79.755, 29.972, -78.215]
  Call Extruder(262.89466)
  MoveL 11414 to (239.41, 155.44, 153.89) mm, rotated rx 180 ry 0 rz 180 deg; joints [-29.466, 13.778, 70.365, 79.761, 29.992, -78.219]
  MoveL 11415 to (239.41, 155.44, 153.89) mm, rotated rx 180 ry 0 rz 180 deg; joints [-29.466, 13.778, 70.365, 79.761, 29.992, -78.219]
  Call Extruder(263.07662)
  MoveL 11416 to (239.29, 155.73, 153.89) mm, rotated rx -180 ry 0 rz 180 deg; joints [-29.499, 13.784, 70.356, 79.771, 30.024, -78.228]
  MoveL 11417 to (239.29, 155.73, 153.89) mm, rotated rx -180 ry 0 rz 180 deg; joints [-29.499, 13.784, 70.356, 79.771, 30.024, -78.228]
  Call Extruder(263.25933)
  MoveL 11418 to (239.16, 156.02, 153.89) mm, rotated rx 180 ry 0 rz 180 deg; joints [-29.531, 13.791, 70.348, 79.782, 30.055, -78.236]
  MoveL 11419 to (239.16, 156.02, 153.89) mm, rotated rx 180 ry 0 rz 180 deg; joints [-29.531, 13.791, 70.348, 79.782, 30.055, -78.236]
  Call Extruder(263.42975)
  MoveL 11420 to (239.05, 156.29, 153.89) mm, rotated rx 180 ry 0 rz 180 deg; joints [-29.561, 13.797, 70.341, 79.792, 30.085, -78.244]
  MoveL 11421 to (239.05, 156.29, 153.89) mm, rotated rx 180 ry 0 rz 180 deg; joints [-29.561, 13.797, 70.341, 79.792, 30.085, -78.244]
  Call Extruder(263.58776)
  MoveL 11422 to (238.94, 156.54, 153.89) mm, rotated rx 180 ry 0 rz 180 deg; joints [-29.589, 13.802, 70.334, 79.801, 30.112, -78.251]
  MoveL 11423 to (238.94, 156.54, 153.89) mm, rotated rx 180 ry 0 rz 180 deg; joints [-29.589, 13.802, 70.334, 79.801, 30.112, -78.251]
  Call Extruder(263.74638)
  MoveL 11424 to (238.84, 156.79, 153.89) mm, rotated rx 180 ry 0 rz 180 deg; joints [-29.617, 13.808, 70.328, 79.811, 30.14, -78.259]
  MoveL 11425 to (238.84, 156.79, 153.89) mm, rotated rx 180 ry 0 rz 180 deg; joints [-29.617, 13.808, 70.328, 79.811, 30.14, -78.259]
  Call Extruder(263.95255)
  MoveL 11426 to (238.66, 157.09, 153.89) mm, rotated rx 180 ry 0 rz 180 deg; joints [-29.653, 13.807, 70.328, 79.825, 30.175, -78.272]
  MoveL 11427 to (238.66, 157.09, 153.89) mm, rotated rx 180 ry 0 rz 180 deg; joints [-29.653, 13.807, 70.328, 79.825, 30.175, -78.272]
  Call Extruder(264.15949)
  MoveL 11428 to (238.49, 157.4, 153.89) mm, rotated rx 180 ry 0 rz 180 deg; joints [-29.689, 13.807, 70.329, 79.84, 30.211, -78.285]
  MoveL 11429 to (238.49, 157.4, 153.89) mm, rotated rx 180 ry 0 rz 180 deg; joints [-29.689, 13.807, 70.329, 79.84, 30.211, -78.285]
  Call Extruder(264.36722)
  MoveL 11430 to (238.31, 157.7, 153.89) mm, rotated rx 180 ry 0 rz 180 deg; joints [-29.725, 13.807, 70.329, 79.855, 30.246, -78.297]
  MoveL 11431 to (238.31, 157.7, 153.89) mm, rotated rx 180 ry 0 rz 180 deg; joints [-29.725, 13.807, 70.329, 79.855, 30.246, -78.297]
  Call Extruder(264.57572)
  MoveL 11432 to (238.13, 158.01, 153.89) mm, rotated rx 180 ry 0 rz 180 deg; joints [-29.761, 13.806, 70.329, 79.869, 30.282, -78.31]
  MoveL 11433 to (238.13, 158.01, 153.89) mm, rotated rx 180 ry 0 rz 180 deg; joints [-29.761, 13.806, 70.329, 79.869, 30.282, -78.31]
  Call Extruder(264.75269)
  MoveL 11434 to (237.96, 158.25, 153.89) mm, rotated rx -180 ry 0 rz -180 deg; joints [-29.792, 13.801, 70.336, 79.884, 30.311, -78.323]
  MoveL 11435 to (237.96, 158.25, 153.89) mm, rotated rx -180 ry 0 rz -180 deg; joints [-29.792, 13.801, 70.336, 79.884, 30.311, -78.323]
  Call Extruder(265.08090)
  MoveL 11436 to (237.64, 158.69, 153.89) mm, rotated rx 180 ry 0 rz -180 deg; joints [-29.848, 13.791, 70.349, 79.91, 30.366, -78.347]
  MoveL 11437 to (237.64, 158.69, 153.89) mm, rotated rx 180 ry 0 rz -180 deg; joints [-29.848, 13.791, 70.349, 79.91, 30.366, -78.347]
  Call Extruder(265.41030)
  MoveL 11438 to (237.32, 159.14, 153.89) mm, rotated rx 180 ry 0 rz 180 deg; joints [-29.904, 13.78, 70.361, 79.936, 30.421, -78.371]
  Call Extruder(266.28192)
  MoveL 11439 to (236.35, 160.23, 153.89) mm, rotated rx 180 ry 0 rz 180 deg; joints [-30.051, 13.729, 70.424, 80.013, 30.563, -78.443]
  Call Extruder(267.07895)
  MoveL 11440 to (235.35, 161.1, 153.89) mm, rotated rx 180 ry 0 rz 180 deg; joints [-30.182, 13.655, 70.514, 80.092, 30.687, -78.518]
  Call Extruder(267.24365)
  MoveL 11441 to (235.13, 161.27, 153.89) mm, rotated rx 180 ry 0 rz 180 deg; joints [-30.208, 13.635, 70.538, 80.109, 30.712, -78.535]
  MoveL 11442 to (235.13, 161.27, 153.89) mm, rotated rx 180 ry 0 rz 180 deg; joints [-30.208, 13.635, 70.538, 80.109, 30.712, -78.535]
  Call Extruder(267.57190)
  MoveL 11443 to (234.69, 161.59, 153.89) mm, rotated rx 180 ry 0 rz -180 deg; joints [-30.259, 13.596, 70.586, 80.143, 30.762, -78.569]
  MoveL 11444 to (234.69, 161.59, 153.89) mm, rotated rx 180 ry 0 rz -180 deg; joints [-30.259, 13.596, 70.586, 80.143, 30.762, -78.569]
  Call Extruder(267.89900)
  MoveL 11445 to (234.24, 161.91, 153.89) mm, rotated rx 180 ry 0 rz 180 deg; joints [-30.311, 13.558, 70.633, 80.177, 30.811, -78.602]
  MoveL 11446 to (234.24, 161.91, 153.89) mm, rotated rx 180 ry 0 rz 180 deg; joints [-30.311, 13.558, 70.633, 80.177, 30.811, -78.602]
  Call Extruder(268.03352)
  MoveL 11447 to (234.05, 162.03, 153.89) mm, rotated rx 180 ry 0 rz -180 deg; joints [-30.332, 13.538, 70.657, 80.192, 30.83, -78.617]
  MoveL 11448 to (234.05, 162.03, 153.89) mm, rotated rx 180 ry 0 rz -180 deg; joints [-30.332, 13.538, 70.657, 80.192, 30.83, -78.617]
  Call Extruder(268.24883)
  MoveL 11449 to (233.73, 162.21, 153.89) mm, rotated rx -180 ry 0 rz -180 deg; joints [-30.364, 13.506, 70.695, 80.216, 30.861, -78.641]
  MoveL 11450 to (233.73, 162.21, 153.89) mm, rotated rx -180 ry 0 rz -180 deg; joints [-30.364, 13.506, 70.695, 80.216, 30.861, -78.641]
  Call Extruder(268.46330)
  MoveL 11451 to (233.41, 162.39, 153.89) mm, rotated rx 180 ry 0 rz 180 deg; joints [-30.397, 13.475, 70.734, 80.24, 30.892, -78.665]
  MoveL 11452 to (233.41, 162.39, 153.89) mm, rotated rx 180 ry 0 rz 180 deg; joints [-30.397, 13.475, 70.734, 80.24, 30.892, -78.665]
  Call Extruder(268.67694)
  MoveL 11453 to (233.1, 162.57, 153.89) mm, rotated rx -180 ry 0 rz 180 deg; joints [-30.43, 13.443, 70.772, 80.263, 30.923, -78.689]
  MoveL 11454 to (233.1, 162.57, 153.89) mm, rotated rx -180 ry 0 rz 180 deg; joints [-30.43, 13.443, 70.772, 80.263, 30.923, -78.689]
  Call Extruder(268.85614)
  MoveL 11455 to (232.83, 162.71, 153.89) mm, rotated rx 180 ry 0 rz 180 deg; joints [-30.457, 13.414, 70.807, 80.284, 30.948, -78.709]
  MoveL 11456 to (232.83, 162.71, 153.89) mm, rotated rx 180 ry 0 rz 180 deg; joints [-30.457, 13.414, 70.807, 80.284, 30.948, -78.709]
  Call Extruder(269.00184)
  MoveL 11457 to (232.6, 162.81, 153.89) mm, rotated rx 180 ry 0 rz -180 deg; joints [-30.477, 13.388, 70.839, 80.301, 30.968, -78.727]
  MoveL 11458 to (232.6, 162.81, 153.89) mm, rotated rx 180 ry 0 rz -180 deg; joints [-30.477, 13.388, 70.839, 80.301, 30.968, -78.727]
  Call Extruder(269.14703)
  MoveL 11459 to (232.37, 162.91, 153.89) mm, rotated rx 180 ry 0 rz 180 deg; joints [-30.498, 13.362, 70.87, 80.318, 30.987, -78.744]
  MoveL 11460 to (232.37, 162.91, 153.89) mm, rotated rx 180 ry 0 rz 180 deg; joints [-30.498, 13.362, 70.87, 80.318, 30.987, -78.744]
  Call Extruder(269.32977)
  MoveL 11461 to (232.08, 163.03, 153.89) mm, rotated rx 180 ry 0 rz 180 deg; joints [-30.524, 13.329, 70.911, 80.34, 31.012, -78.767]
  MoveL 11462 to (232.08, 163.03, 153.89) mm, rotated rx 180 ry 0 rz 180 deg; joints [-30.524, 13.329, 70.911, 80.34, 31.012, -78.767]
  Call Extruder(269.51175)
  MoveL 11463 to (231.78, 163.15, 153.89) mm, rotated rx 180 ry 0 rz 180 deg; joints [-30.551, 13.296, 70.951, 80.361, 31.036, -78.789]
  MoveL 11464 to (231.78, 163.15, 153.89) mm, rotated rx 180 ry 0 rz 180 deg; joints [-30.551, 13.296, 70.951, 80.361, 31.036, -78.789]
  Call Extruder(269.65909)
  MoveL 11465 to (231.54, 163.24, 153.89) mm, rotated rx 180 ry 0 rz 180 deg; joints [-30.571, 13.268, 70.985, 80.379, 31.055, -78.807]
  MoveL 11466 to (231.54, 163.24, 153.89) mm, rotated rx 180 ry 0 rz 180 deg; joints [-30.571, 13.268, 70.985, 80.379, 31.055, -78.807]
  Call Extruder(269.77231)
  MoveL 11467 to (231.35, 163.3, 153.89) mm, rotated rx 180 ry 0 rz 180 deg; joints [-30.587, 13.245, 71.013, 80.392, 31.07, -78.821]
  MoveL 11468 to (231.35, 163.3, 153.89) mm, rotated rx 180 ry 0 rz 180 deg; joints [-30.587, 13.245, 71.013, 80.392, 31.07, -78.821]
  Call Extruder(269.88509)
  MoveL 11469 to (231.17, 163.36, 153.89) mm, rotated rx 180 ry 0 rz 180 deg; joints [-30.602, 13.222, 71.041, 80.406, 31.084, -78.835]
  MoveL 11470 to (231.17, 163.36, 153.89) mm, rotated rx 180 ry 0 rz 180 deg; joints [-30.602, 13.222, 71.041, 80.406, 31.084, -78.835]
  Call Extruder(269.99742)
  MoveL 11471 to (230.98, 163.42, 153.89) mm, rotated rx 180 ry 0 rz -180 deg; joints [-30.618, 13.199, 71.069, 80.42, 31.098, -78.849]
  MoveL 11472 to (230.98, 163.42, 153.89) mm, rotated rx 180 ry 0 rz -180 deg; joints [-30.618, 13.199, 71.069, 80.42, 31.098, -78.849]
  Call Extruder(270.10931)
  MoveL 11473 to (230.79, 163.48, 153.89) mm, rotated rx 180 ry 0 rz 180 deg; joints [-30.633, 13.176, 71.096, 80.434, 31.113, -78.864]
  MoveL 11474 to (230.79, 163.48, 153.89) mm, rotated rx 180 ry 0 rz 180 deg; joints [-30.633, 13.176, 71.096, 80.434, 31.113, -78.864]
  Call Extruder(270.23072)
  MoveL 11475 to (230.58, 163.55, 153.89) mm, rotated rx -180 ry 0 rz 180 deg; joints [-30.65, 13.151, 71.127, 80.448, 31.128, -78.879]
  MoveL 11476 to (230.58, 163.55, 153.89) mm, rotated rx -180 ry 0 rz 180 deg; joints [-30.65, 13.151, 71.127, 80.448, 31.128, -78.879]
  Call Extruder(270.36153)
  MoveL 11477 to (230.36, 163.62, 153.89) mm, rotated rx 180 ry 0 rz -180 deg; joints [-30.668, 13.123, 71.16, 80.465, 31.145, -78.896]
  MoveL 11478 to (230.36, 163.62, 153.89) mm, rotated rx 180 ry 0 rz -180 deg; joints [-30.668, 13.123, 71.16, 80.465, 31.145, -78.896]
  Call Extruder(270.49178)
  MoveL 11479 to (230.14, 163.68, 153.89) mm, rotated rx 180 ry 0 rz -180 deg; joints [-30.685, 13.096, 71.193, 80.481, 31.161, -78.913]
  MoveL 11480 to (230.14, 163.68, 153.89) mm, rotated rx 180 ry 0 rz -180 deg; joints [-30.685, 13.096, 71.193, 80.481, 31.161, -78.913]
  Call Extruder(270.62146)
  MoveL 11481 to (229.91, 163.75, 153.89) mm, rotated rx -180 ry 0 rz 180 deg; joints [-30.703, 13.068, 71.227, 80.497, 31.178, -78.929]
  MoveL 11482 to (229.91, 163.75, 153.89) mm, rotated rx -180 ry 0 rz 180 deg; joints [-30.703, 13.068, 71.227, 80.497, 31.178, -78.929]
  Call Extruder(270.75058)
  MoveL 11483 to (229.69, 163.82, 153.89) mm, rotated rx 180 ry 0 rz 180 deg; joints [-30.721, 13.04, 71.26, 80.513, 31.195, -78.946]
  MoveL 11484 to (229.69, 163.82, 153.89) mm, rotated rx 180 ry 0 rz 180 deg; joints [-30.721, 13.04, 71.26, 80.513, 31.195, -78.946]
  Call Extruder(270.86565)
  MoveL 11485 to (229.48, 163.86, 153.89) mm, rotated rx -180 ry 0 rz 180 deg; joints [-30.736, 13.014, 71.292, 80.527, 31.208, -78.961]
  MoveL 11486 to (229.48, 163.86, 153.89) mm, rotated rx -180 ry 0 rz 180 deg; joints [-30.736, 13.014, 71.292, 80.527, 31.208, -78.961]
  Call Extruder(270.98027)
  MoveL 11487 to (229.28, 163.91, 153.89) mm, rotated rx 180 ry 0 rz 180 deg; joints [-30.751, 12.987, 71.324, 80.542, 31.222, -78.976]
  MoveL 11488 to (229.28, 163.91, 153.89) mm, rotated rx 180 ry 0 rz 180 deg; joints [-30.751, 12.987, 71.324, 80.542, 31.222, -78.976]
